LIN {X 0,Y 433.075,Z 406.489,A -85,B 0,C 180,E1 21289.378,E2 21289.378} C_VEL
LIN {X 0,Y 433.196,Z 405.398,A -85,B 0,C 180,E1 21287.416,E2 21287.416} C_VEL
LIN {X 0,Y 433.474,Z 402.273,A -85,B 0,C 180,E1 21285.29,E2 21285.29} C_VEL
LIN {X 0,Y 433.894,Z 397.242,A -85,B 0,C 180,E1 21283.265,E2 21283.265} C_VEL
LIN {X 0,Y 434.433,Z 391.164,A -85,B 0,C 180,E1 21281.517,E2 21281.517} C_VEL
LIN {X 0,Y 435.19,Z 382.602,A -85,B 0,C 180,E1 21279.675,E2 21279.675} C_VEL
LIN {X 0,Y 436.03,Z 373.053,A -85,B 0,C 180,E1 21278.086,E2 21278.086} C_VEL
LIN {X 0,Y 436.996,Z 361.523,A -85,B 0,C 180,E1 21276.573,E2 21276.573} C_VEL
LIN {X 0,Y 437.95,Z 348.916,A -85,B 0,C 180,E1 21275.283,E2 21275.283} C_VEL
LIN {X 0,Y 438.832,Z 335.315,A -85,B 0,C 180,E1 21274.2,E2 21274.2} C_VEL
LIN {X 0,Y 439.584,Z 321.029,A -85,B 0,C 180,E1 21273.335,E2 21273.335} C_VEL
LIN {X 0,Y 440.16,Z 305.307,A -85,B 0,C 180,E1 21272.665,E2 21272.665} C_VEL
LIN {X 0,Y 440.515,Z 289.237,A -85,B 0,C 180,E1 21272.235,E2 21272.235} C_VEL
LIN {X 0,Y 442.617,Z 196.385,A -85,B 0,C 180,E1 21270.394,E2 21270.394} C_VEL
LIN {X 0,Y 438.448,Z 173.54,A -85,B 0,C 180,E1 21269.604,E2 21269.604} C_VEL
LIN {X 0,Y 440.626,Z 144.172,A -85,B 0,C 180,E1 21265.541,E2 21265.541} C_VEL
LIN {X 0,Y 442.984,Z 116.613,A -85,B 0,C 180,E1 21261.65,E2 21261.65} C_VEL
LIN {X 0,Y 444.119,Z 103.787,A -85,B 0,C 180,E1 21259.806,E2 21259.806} C_VEL
LIN {X 0,Y 440.05,Z 88.666,A -85,B 0,C 180,E1 21257.044,E2 21257.044} C_VEL
LIN {X 0,Y 435.296,Z 73.845,A -85,B 0,C 180,E1 21254.092,E2 21254.092} C_VEL
LIN {X 0,Y 433.235,Z 67.94,A -85,B 0,C 180,E1 21252.767,E2 21252.767} C_VEL
LIN {X 0,Y 433.212,Z 67.828,A -85,B 0,C 180,E1 21249.03,E2 21249.03} C_VEL
LIN {X 0,Y 433.209,Z 67.837,A -85,B 0,C 180,E1 21245.297,E2 21245.297} C_VEL
LIN {X 0,Y 433.214,Z 67.833,A -85,B 0,C 180,E1 21241.587,E2 21241.587} C_VEL
LIN {X 0,Y 433.223,Z 67.833,A -85,B 0,C 180,E1 21237.924,E2 21237.924} C_VEL
LIN {X 0,Y 433.235,Z 67.831,A -85,B 0,C 180,E1 21234.172,E2 21234.172} C_VEL
LIN {X 0,Y 433.245,Z 67.831,A -85,B 0,C 180,E1 21230.435,E2 21230.435} C_VEL
LIN {X 0,Y 433.25,Z 67.833,A -85,B 0,C 180,E1 21226.657,E2 21226.657} C_VEL
LIN {X 0,Y 433.243,Z 67.831,A -85,B 0,C 180,E1 21222.818,E2 21222.818} C_VEL
LIN {X 0,Y 433.231,Z 67.83,A -85,B 0,C 180,E1 21219.04,E2 21219.04} C_VEL
LIN {X 0,Y 433.214,Z 67.833,A -85,B 0,C 180,E1 21215.308,E2 21215.308} C_VEL
LIN {X 0,Y 433.2,Z 67.836,A -85,B 0,C 180,E1 21211.611,E2 21211.611} C_VEL
LIN {X 0,Y 433.191,Z 67.837,A -85,B 0,C 180,E1 21207.896,E2 21207.896} C_VEL
LIN {X 0,Y 433.19,Z 67.836,A -85,B 0,C 180,E1 21204.108,E2 21204.108} C_VEL
LIN {X 0,Y 433.187,Z 67.839,A -85,B 0,C 180,E1 21200.256,E2 21200.256} C_VEL
LIN {X 0,Y 433.192,Z 67.835,A -85,B 0,C 180,E1 21196.542,E2 21196.542} C_VEL
LIN {X 0,Y 433.211,Z 67.832,A -85,B 0,C 180,E1 21192.912,E2 21192.912} C_VEL
LIN {X 0,Y 433.263,Z 68.081,A -85,B 0,C 180,E1 21191.105,E2 21191.105} C_VEL
LIN {X 0,Y 438.845,Z 82.472,A -85,B 0,C 180,E1 21188.603,E2 21188.603} C_VEL
LIN {X 0,Y 444.549,Z 98.48,A -85,B 0,C 180,E1 21186.153,E2 21186.153} C_VEL
LIN {X 0,Y 447.389,Z 107.578,A -85,B 0,C 180,E1 21184.895,E2 21184.895} C_VEL
LIN {X 0,Y 443.251,Z 148.715,A -85,B 0,C 180,E1 21180.876,E2 21180.876} C_VEL
LIN {X 0,Y 442.316,Z 161.133,A -85,B 0,C 180,E1 21179.733,E2 21179.733} C_VEL
LIN {X 0,Y 444.429,Z 180.599,A -85,B 0,C 180,E1 21179.248,E2 21179.248} C_VEL
LIN {X 0,Y 442.001,Z 357.769,A -85,B 0,C 180,E1 21176.343,E2 21176.343} C_VEL
LIN {X 0,Y 441.177,Z 376.273,A -85,B 0,C 180,E1 21175.815,E2 21175.815} C_VEL
LIN {X 0,Y 440.124,Z 394.053,A -85,B 0,C 180,E1 21175.068,E2 21175.068} C_VEL
LIN {X 0,Y 438.871,Z 411.762,A -85,B 0,C 180,E1 21174.068,E2 21174.068} C_VEL
LIN {X 0,Y 437.522,Z 428.981,A -85,B 0,C 180,E1 21172.82,E2 21172.82} C_VEL
LIN {X 0,Y 436.208,Z 445.015,A -85,B 0,C 180,E1 21171.375,E2 21171.375} C_VEL
LIN {X 0,Y 435.015,Z 459.816,A -85,B 0,C 180,E1 21169.748,E2 21169.748} C_VEL
LIN {X 0,Y 433.995,Z 473.598,A -85,B 0,C 180,E1 21167.92,E2 21167.92} C_VEL
LIN {X 0,Y 433.196,Z 485.958,A -85,B 0,C 180,E1 21165.943,E2 21165.943} C_VEL
LIN {X 0,Y 432.671,Z 497.125,A -85,B 0,C 180,E1 21163.771,E2 21163.771} C_VEL
LIN {X 0,Y 432.402,Z 506.213,A -85,B 0,C 180,E1 21161.606,E2 21161.606} C_VEL
LIN {X 0,Y 432.351,Z 513.891,A -85,B 0,C 180,E1 21159.317,E2 21159.317} C_VEL
LIN {X 0,Y 432.443,Z 519.752,A -85,B 0,C 180,E1 21157.04,E2 21157.04} C_VEL
LIN {X 0,Y 432.595,Z 524.105,A -85,B 0,C 180,E1 21154.641,E2 21154.641} C_VEL
LIN {X 0,Y 432.715,Z 526.668,A -85,B 0,C 180,E1 21152.252,E2 21152.252} C_VEL
LIN {X 0,Y 432.765,Z 527.51,A -85,B 0,C 180,E1 21150.001,E2 21150.001} C_VEL
LIN {X 0,Y 432.693,Z 526.696,A -85,B 0,C 180,E1 21147.617,E2 21147.617} C_VEL
LIN {X 0,Y 432.564,Z 524.137,A -85,B 0,C 180,E1 21145.228,E2 21145.228} C_VEL
LIN {X 0,Y 432.407,Z 519.767,A -85,B 0,C 180,E1 21142.828,E2 21142.828} C_VEL
LIN {X 0,Y 432.328,Z 513.478,A -85,B 0,C 180,E1 21140.416,E2 21140.416} C_VEL
LIN {X 0,Y 432.413,Z 505.642,A -85,B 0,C 180,E1 21138.125,E2 21138.125} C_VEL
LIN {X 0,Y 432.721,Z 496.365,A -85,B 0,C 180,E1 21135.96,E2 21135.96} C_VEL
LIN {X 0,Y 433.259,Z 485.712,A -85,B 0,C 180,E1 21133.924,E2 21133.924} C_VEL
LIN {X 0,Y 434.052,Z 473.719,A -85,B 0,C 180,E1 21132.022,E2 21132.022} C_VEL
LIN {X 0,Y 435.095,Z 459.77,A -85,B 0,C 180,E1 21130.188,E2 21130.188} C_VEL
LIN {X 0,Y 436.299,Z 444.783,A -85,B 0,C 180,E1 21128.562,E2 21128.562} C_VEL
LIN {X 0,Y 437.586,Z 428.819,A -85,B 0,C 180,E1 21127.144,E2 21127.144} C_VEL
LIN {X 0,Y 438.881,Z 411.866,A -85,B 0,C 180,E1 21125.935,E2 21125.935} C_VEL
LIN {X 0,Y 440.066,Z 394.468,A -85,B 0,C 180,E1 21124.967,E2 21124.967} C_VEL
LIN {X 0,Y 441.097,Z 376.307,A -85,B 0,C 180,E1 21124.217,E2 21124.217} C_VEL
LIN {X 0,Y 441.882,Z 357.278,A -85,B 0,C 180,E1 21123.69,E2 21123.69} C_VEL
LIN {X 0,Y 444.228,Z 168.638,A -85,B 0,C 180,E1 21120.613,E2 21120.613} C_VEL
LIN {X 0,Y 443.59,Z 156.452,A -85,B 0,C 180,E1 21120.348,E2 21120.348} C_VEL
LIN {X 0,Y 446.644,Z 101.681,A -85,B 0,C 180,E1 21117.321,E2 21117.321} C_VEL
LIN {X 0,Y 436.652,Z 76.57,A -85,B 0,C 180,E1 21115.06,E2 21115.06} C_VEL
LIN {X 0,Y 433.339,Z 68.369,A -85,B 0,C 180,E1 21114.246,E2 21114.246} C_VEL
LIN {X 0,Y 433.254,Z 67.833,A -85,B 0,C 180,E1 21113.952,E2 21113.952} C_VEL
LIN {X 0,Y 433.255,Z 67.829,A -85,B 0,C 180,E1 21110.094,E2 21110.094} C_VEL
LIN {X 0,Y 433.255,Z 67.829,A -85,B 0,C 180,E1 21106.247,E2 21106.247} C_VEL
LIN {X 0,Y 433.258,Z 67.83,A -85,B 0,C 180,E1 21102.366,E2 21102.366} C_VEL
LIN {X 0,Y 433.259,Z 67.826,A -85,B 0,C 180,E1 21098.528,E2 21098.528} C_VEL
LIN {X 0,Y 433.259,Z 67.822,A -85,B 0,C 180,E1 21094.751,E2 21094.751} C_VEL
LIN {X 0,Y 433.26,Z 67.824,A -85,B 0,C 180,E1 21090.857,E2 21090.857} C_VEL
LIN {X 0,Y 433.256,Z 67.822,A -85,B 0,C 180,E1 21087.03,E2 21087.03} C_VEL
LIN {X 0,Y 433.252,Z 67.819,A -85,B 0,C 180,E1 21083.243,E2 21083.243} C_VEL
LIN {X 0,Y 433.24,Z 67.823,A -85,B 0,C 180,E1 21079.55,E2 21079.55} C_VEL
LIN {X 0,Y 433.235,Z 67.827,A -85,B 0,C 180,E1 21075.771,E2 21075.771} C_VEL
LIN {X 0,Y 433.234,Z 67.83,A -85,B 0,C 180,E1 21071.988,E2 21071.988} C_VEL
LIN {X 0,Y 433.232,Z 67.829,A -85,B 0,C 180,E1 21068.093,E2 21068.093} C_VEL
LIN {X 0,Y 433.231,Z 67.825,A -85,B 0,C 180,E1 21064.235,E2 21064.235} C_VEL
LIN {X 0,Y 433.229,Z 67.822,A -85,B 0,C 180,E1 21060.396,E2 21060.396} C_VEL
LIN {X 0,Y 433.236,Z 67.829,A -85,B 0,C 180,E1 21056.692,E2 21056.692} C_VEL
LIN {X 0,Y 433.244,Z 67.833,A -85,B 0,C 180,E1 21052.902,E2 21052.902} C_VEL
LIN {X 0,Y 433.247,Z 67.829,A -85,B 0,C 180,E1 21049.091,E2 21049.091} C_VEL
LIN {X 0,Y 433.257,Z 67.824,A -85,B 0,C 180,E1 21045.294,E2 21045.294} C_VEL
LIN {X 0,Y 433.256,Z 67.824,A -85,B 0,C 180,E1 21041.429,E2 21041.429} C_VEL
LIN {X 0,Y 433.264,Z 67.81,A -85,B 0,C 180,E1 21037.618,E2 21037.618} C_VEL
LIN {X 0,Y 433.258,Z 67.826,A -85,B 0,C 180,E1 21033.698,E2 21033.698} C_VEL
LIN {X 0,Y 433.26,Z 67.809,A -85,B 0,C 180,E1 21029.926,E2 21029.926} C_VEL
LIN {X 0,Y 433.254,Z 67.83,A -85,B 0,C 180,E1 21026.048,E2 21026.048} C_VEL
LIN {X 0,Y 433.239,Z 67.832,A -85,B 0,C 180,E1 21022.295,E2 21022.295} C_VEL
LIN {X 0,Y 433.222,Z 67.83,A -85,B 0,C 180,E1 21018.595,E2 21018.595} C_VEL
LIN {X 0,Y 433.213,Z 67.834,A -85,B 0,C 180,E1 21014.882,E2 21014.882} C_VEL
LIN {X 0,Y 433.204,Z 67.837,A -85,B 0,C 180,E1 21011.13,E2 21011.13} C_VEL
LIN {X 0,Y 433.261,Z 68.1,A -85,B 0,C 180,E1 21008.676,E2 21008.676} C_VEL
LIN {X 0,Y 438.519,Z 85.922,A -85,B 0,C 180,E1 21006.292,E2 21006.292} C_VEL
LIN {X 0,Y 440.008,Z 92.89,A -85,B 0,C 180,E1 21005.41,E2 21005.41} C_VEL
LIN {X 0,Y 439.529,Z 126.207,A -85,B 0,C 180,E1 21001.699,E2 21001.699} C_VEL
LIN {X 0,Y 438.985,Z 159.572,A -85,B 0,C 180,E1 20997.981,E2 20997.981} C_VEL
LIN {X 0,Y 438.678,Z 192.545,A -85,B 0,C 180,E1 20994.455,E2 20994.455} C_VEL
LIN {X 0,Y 439.206,Z 197.779,A -85,B 0,C 180,E1 20994.332,E2 20994.332} C_VEL
LIN {X 0,Y 438.077,Z 288.666,A -85,B 0,C 180,E1 20992.826,E2 20992.826} C_VEL
LIN {X 0,Y 437.082,Z 296.35,A -85,B 0,C 180,E1 20992.742,E2 20992.742} C_VEL
LIN {X 0,Y 432.175,Z 312.347,A -85,B 0,C 180,E1 20992.59,E2 20992.59} C_VEL
LIN {X 0,Y 430.641,Z 319.881,A -85,B 0,C 180,E1 20992.382,E2 20992.382} C_VEL
LIN {X 0,Y 430.425,Z 322.967,A -85,B 0,C 180,E1 20992.254,E2 20992.254} C_VEL
LIN {X 0,Y 430.017,Z 337.032,A -85,B 0,C 180,E1 20991.481,E2 20991.481} C_VEL
LIN {X 0,Y 429.406,Z 349.966,A -85,B 0,C 180,E1 20990.512,E2 20990.512} C_VEL
LIN {X 0,Y 428.679,Z 362.566,A -85,B 0,C 180,E1 20989.27,E2 20989.27} C_VEL
LIN {X 0,Y 427.886,Z 373.856,A -85,B 0,C 180,E1 20987.824,E2 20987.824} C_VEL
LIN {X 0,Y 427.151,Z 383.064,A -85,B 0,C 180,E1 20986.312,E2 20986.312} C_VEL
LIN {X 0,Y 426.501,Z 390.945,A -85,B 0,C 180,E1 20984.665,E2 20984.665} C_VEL
LIN {X 0,Y 425.929,Z 397.841,A -85,B 0,C 180,E1 20982.747,E2 20982.747} C_VEL
LIN {X 0,Y 425.507,Z 402.946,A -85,B 0,C 180,E1 20980.697,E2 20980.697} C_VEL
LIN {X 0,Y 425.241,Z 406.026,A -85,B 0,C 180,E1 20978.654,E2 20978.654} C_VEL
LIN {X 0,Y 425.112,Z 407.274,A -85,B 0,C 180,E1 20976.617,E2 20976.617} C_VEL
LIN {X 0,Y 425.103,Z 406.761,A -85,B 0,C 180,E1 20974.586,E2 20974.586} C_VEL
LIN {X 0,Y 425.219,Z 404.234,A -85,B 0,C 180,E1 20972.425,E2 20972.425} C_VEL
LIN {X 0,Y 425.464,Z 399.9,A -85,B 0,C 180,E1 20970.403,E2 20970.403} C_VEL
LIN {X 0,Y 425.825,Z 393.939,A -85,B 0,C 180,E1 20968.519,E2 20968.519} C_VEL
LIN {X 0,Y 426.31,Z 386.487,A -85,B 0,C 180,E1 20966.772,E2 20966.772} C_VEL
LIN {X 0,Y 426.895,Z 377.575,A -85,B 0,C 180,E1 20965.162,E2 20965.162} C_VEL
LIN {X 0,Y 427.565,Z 366.546,A -85,B 0,C 180,E1 20963.622,E2 20963.622} C_VEL
LIN {X 0,Y 428.158,Z 354.829,A -85,B 0,C 180,E1 20962.35,E2 20962.35} C_VEL
LIN {X 0,Y 428.687,Z 342.994,A -85,B 0,C 180,E1 20961.347,E2 20961.347} C_VEL
LIN {X 0,Y 429.131,Z 329.341,A -85,B 0,C 180,E1 20960.477,E2 20960.477} C_VEL
LIN {X 0,Y 429.327,Z 314.736,A -85,B 0,C 180,E1 20959.825,E2 20959.825} C_VEL
LIN {X 0,Y 429.329,Z 299.926,A -85,B 0,C 180,E1 20959.423,E2 20959.423} C_VEL
LIN {X 0,Y 430.516,Z 189.532,A -85,B 0,C 180,E1 20957.56,E2 20957.56} C_VEL
LIN {X 0,Y 431.081,Z 159.552,A -85,B 0,C 180,E1 20955.629,E2 20955.629} C_VEL
LIN {X 0,Y 431.654,Z 130.351,A -85,B 0,C 180,E1 20953.653,E2 20953.653} C_VEL
LIN {X 0,Y 432.206,Z 129.541,A -85,B 0,C 180,E1 20953.433,E2 20953.433} C_VEL
LIN {X 0,Y 434.053,Z 130.583,A -85,B 0,C 180,E1 20953.161,E2 20953.161} C_VEL
LIN {X 0,Y 431.916,Z 170.793,A -85,B 0,C 180,E1 20949.928,E2 20949.928} C_VEL
LIN {X 0,Y 433.654,Z 190.939,A -85,B 0,C 180,E1 20949.44,E2 20949.44} C_VEL
LIN {X 0,Y 431.591,Z 296.803,A -85,B 0,C 180,E1 20947.438,E2 20947.438} C_VEL
LIN {X 0,Y 431.154,Z 313.161,A -85,B 0,C 180,E1 20946.871,E2 20946.871} C_VEL
LIN {X 0,Y 430.489,Z 328.565,A -85,B 0,C 180,E1 20946.064,E2 20946.064} C_VEL
LIN {X 0,Y 429.718,Z 342.273,A -85,B 0,C 180,E1 20945.092,E2 20945.092} C_VEL
LIN {X 0,Y 428.833,Z 355.782,A -85,B 0,C 180,E1 20943.853,E2 20943.853} C_VEL
LIN {X 0,Y 427.907,Z 368.637,A -85,B 0,C 180,E1 20942.324,E2 20942.324} C_VEL
LIN {X 0,Y 427.079,Z 379.255,A -85,B 0,C 180,E1 20940.705,E2 20940.705} C_VEL
LIN {X 0,Y 426.438,Z 387.604,A -85,B 0,C 180,E1 20939.103,E2 20939.103} C_VEL
LIN {X 0,Y 425.856,Z 395.37,A -85,B 0,C 180,E1 20937.155,E2 20937.155} C_VEL
LIN {X 0,Y 425.493,Z 400.746,A -85,B 0,C 180,E1 20935.333,E2 20935.333} C_VEL
LIN {X 0,Y 425.248,Z 404.826,A -85,B 0,C 180,E1 20933.3,E2 20933.3} C_VEL
LIN {X 0,Y 425.139,Z 407.07,A -85,B 0,C 180,E1 20931.274,E2 20931.274} C_VEL
LIN {X 0,Y 425.165,Z 407.601,A -85,B 0,C 180,E1 20929.173,E2 20929.173} C_VEL
LIN {X 0,Y 425.304,Z 406.351,A -85,B 0,C 180,E1 20927.18,E2 20927.18} C_VEL
LIN {X 0,Y 425.607,Z 403.261,A -85,B 0,C 180,E1 20925.096,E2 20925.096} C_VEL
LIN {X 0,Y 426.062,Z 398.275,A -85,B 0,C 180,E1 20923.071,E2 20923.071} C_VEL
LIN {X 0,Y 426.687,Z 391.722,A -85,B 0,C 180,E1 20921.184,E2 20921.184} C_VEL
LIN {X 0,Y 427.515,Z 383.155,A -85,B 0,C 180,E1 20919.332,E2 20919.332} C_VEL
LIN {X 0,Y 428.437,Z 373.304,A -85,B 0,C 180,E1 20917.694,E2 20917.694} C_VEL
LIN {X 0,Y 429.449,Z 361.862,A -85,B 0,C 180,E1 20916.191,E2 20916.191} C_VEL
LIN {X 0,Y 430.51,Z 348.756,A -85,B 0,C 180,E1 20914.844,E2 20914.844} C_VEL
LIN {X 0,Y 431.43,Z 335.21,A -85,B 0,C 180,E1 20913.769,E2 20913.769} C_VEL
LIN {X 0,Y 432.234,Z 320.637,A -85,B 0,C 180,E1 20912.891,E2 20912.891} C_VEL
LIN {X 0,Y 432.865,Z 304.237,A -85,B 0,C 180,E1 20912.199,E2 20912.199} C_VEL
LIN {X 0,Y 433.284,Z 285.362,A -85,B 0,C 180,E1 20911.729,E2 20911.729} C_VEL
LIN {X 0,Y 435.428,Z 197.571,A -85,B 0,C 180,E1 20909.949,E2 20909.949} C_VEL
LIN {X 0,Y 430.996,Z 173.326,A -85,B 0,C 180,E1 20909.081,E2 20909.081} C_VEL
LIN {X 0,Y 433.342,Z 144.216,A -85,B 0,C 180,E1 20904.976,E2 20904.976} C_VEL
LIN {X 0,Y 435.85,Z 117.318,A -85,B 0,C 180,E1 20901.111,E2 20901.111} C_VEL
LIN {X 0,Y 436.789,Z 106.47,A -85,B 0,C 180,E1 20899.525,E2 20899.525} C_VEL
LIN {X 0,Y 432.67,Z 91.123,A -85,B 0,C 180,E1 20896.652,E2 20896.652} C_VEL
LIN {X 0,Y 428.146,Z 77.113,A -85,B 0,C 180,E1 20893.781,E2 20893.781} C_VEL
LIN {X 0,Y 425.328,Z 68.949,A -85,B 0,C 180,E1 20891.939,E2 20891.939} C_VEL
LIN {X 0,Y 425.321,Z 68.817,A -85,B 0,C 180,E1 20888.109,E2 20888.109} C_VEL
LIN {X 0,Y 425.312,Z 68.82,A -85,B 0,C 180,E1 20884.315,E2 20884.315} C_VEL
LIN {X 0,Y 425.322,Z 68.819,A -85,B 0,C 180,E1 20880.404,E2 20880.404} C_VEL
LIN {X 0,Y 425.308,Z 68.821,A -85,B 0,C 180,E1 20876.496,E2 20876.496} C_VEL
LIN {X 0,Y 425.32,Z 68.819,A -85,B 0,C 180,E1 20872.571,E2 20872.571} C_VEL
LIN {X 0,Y 425.307,Z 68.821,A -85,B 0,C 180,E1 20868.611,E2 20868.611} C_VEL
LIN {X 0,Y 425.311,Z 68.821,A -85,B 0,C 180,E1 20864.734,E2 20864.734} C_VEL
LIN {X 0,Y 425.305,Z 68.819,A -85,B 0,C 180,E1 20860.784,E2 20860.784} C_VEL
LIN {X 0,Y 425.307,Z 68.818,A -85,B 0,C 180,E1 20856.884,E2 20856.884} C_VEL
LIN {X 0,Y 425.3,Z 68.819,A -85,B 0,C 180,E1 20853.001,E2 20853.001} C_VEL
LIN {X 0,Y 425.294,Z 68.82,A -85,B 0,C 180,E1 20849.169,E2 20849.169} C_VEL
LIN {X 0,Y 425.282,Z 68.822,A -85,B 0,C 180,E1 20845.323,E2 20845.323} C_VEL
LIN {X 0,Y 425.272,Z 68.825,A -85,B 0,C 180,E1 20841.529,E2 20841.529} C_VEL
LIN {X 0,Y 425.25,Z 68.827,A -85,B 0,C 180,E1 20837.925,E2 20837.925} C_VEL
LIN {X 0,Y 425.253,Z 68.824,A -85,B 0,C 180,E1 20834.104,E2 20834.104} C_VEL
LIN {X 0,Y 425.296,Z 69.092,A -85,B 0,C 180,E1 20831.982,E2 20831.982} C_VEL
LIN {X 0,Y 430.877,Z 83.146,A -85,B 0,C 180,E1 20829.4,E2 20829.4} C_VEL
LIN {X 0,Y 436.843,Z 99.589,A -85,B 0,C 180,E1 20826.766,E2 20826.766} C_VEL
LIN {X 0,Y 440.209,Z 110.166,A -85,B 0,C 180,E1 20825.235,E2 20825.235} C_VEL
LIN {X 0,Y 435.706,Z 152.651,A -85,B 0,C 180,E1 20821.01,E2 20821.01} C_VEL
LIN {X 0,Y 435.023,Z 161.252,A -85,B 0,C 180,E1 20820.209,E2 20820.209} C_VEL
LIN {X 0,Y 437.229,Z 181.414,A -85,B 0,C 180,E1 20819.693,E2 20819.693} C_VEL
LIN {X 0,Y 434.628,Z 357.34,A -85,B 0,C 180,E1 20816.756,E2 20816.756} C_VEL
LIN {X 0,Y 433.759,Z 375.802,A -85,B 0,C 180,E1 20816.219,E2 20816.219} C_VEL
LIN {X 0,Y 432.644,Z 393.542,A -85,B 0,C 180,E1 20815.459,E2 20815.459} C_VEL
LIN {X 0,Y 431.315,Z 411.168,A -85,B 0,C 180,E1 20814.444,E2 20814.444} C_VEL
LIN {X 0,Y 429.924,Z 427.831,A -85,B 0,C 180,E1 20813.217,E2 20813.217} C_VEL
LIN {X 0,Y 428.548,Z 443.615,A -85,B 0,C 180,E1 20811.776,E2 20811.776} C_VEL
LIN {X 0,Y 427.263,Z 458.477,A -85,B 0,C 180,E1 20810.122,E2 20810.122} C_VEL
LIN {X 0,Y 426.191,Z 471.87,A -85,B 0,C 180,E1 20808.323,E2 20808.323} C_VEL
LIN {X 0,Y 425.295,Z 484.717,A -85,B 0,C 180,E1 20806.247,E2 20806.247} C_VEL
LIN {X 0,Y 424.714,Z 495.919,A -85,B 0,C 180,E1 20804.034,E2 20804.034} C_VEL
LIN {X 0,Y 424.425,Z 505.036,A -85,B 0,C 180,E1 20801.828,E2 20801.828} C_VEL
LIN {X 0,Y 424.371,Z 512.736,A -85,B 0,C 180,E1 20799.494,E2 20799.494} C_VEL
LIN {X 0,Y 424.474,Z 518.615,A -85,B 0,C 180,E1 20797.173,E2 20797.173} C_VEL
LIN {X 0,Y 424.648,Z 522.983,A -85,B 0,C 180,E1 20794.728,E2 20794.728} C_VEL
LIN {X 0,Y 424.776,Z 525.476,A -85,B 0,C 180,E1 20792.429,E2 20792.429} C_VEL
LIN {X 0,Y 424.842,Z 526.401,A -85,B 0,C 180,E1 20790.001,E2 20790.001} C_VEL
LIN {X 0,Y 424.763,Z 525.58,A -85,B 0,C 180,E1 20787.573,E2 20787.573} C_VEL
LIN {X 0,Y 424.613,Z 523.005,A -85,B 0,C 180,E1 20785.138,E2 20785.138} C_VEL
LIN {X 0,Y 424.442,Z 518.61,A -85,B 0,C 180,E1 20782.693,E2 20782.693} C_VEL
LIN {X 0,Y 424.35,Z 512.711,A -85,B 0,C 180,E1 20780.371,E2 20780.371} C_VEL
LIN {X 0,Y 424.428,Z 504.945,A -85,B 0,C 180,E1 20778.037,E2 20778.037} C_VEL
LIN {X 0,Y 424.744,Z 495.736,A -85,B 0,C 180,E1 20775.83,E2 20775.83} C_VEL
LIN {X 0,Y 425.311,Z 485.158,A -85,B 0,C 180,E1 20773.756,E2 20773.756} C_VEL
LIN {X 0,Y 426.145,Z 473.25,A -85,B 0,C 180,E1 20771.818,E2 20771.818} C_VEL
LIN {X 0,Y 427.242,Z 459.383,A -85,B 0,C 180,E1 20769.951,E2 20769.951} C_VEL
LIN {X 0,Y 428.506,Z 444.483,A -85,B 0,C 180,E1 20768.296,E2 20768.296} C_VEL
LIN {X 0,Y 429.926,Z 427.783,A -85,B 0,C 180,E1 20766.786,E2 20766.786} C_VEL
LIN {X 0,Y 431.214,Z 411.814,A -85,B 0,C 180,E1 20765.625,E2 20765.625} C_VEL
LIN {X 0,Y 432.456,Z 394.611,A -85,B 0,C 180,E1 20764.641,E2 20764.641} C_VEL
LIN {X 0,Y 433.541,Z 376.567,A -85,B 0,C 180,E1 20763.874,E2 20763.874} C_VEL
LIN {X 0,Y 434.371,Z 357.859,A -85,B 0,C 180,E1 20763.336,E2 20763.336} C_VEL
LIN {X 0,Y 436.872,Z 168.968,A -85,B 0,C 180,E1 20760.199,E2 20760.199} C_VEL
LIN {X 0,Y 436.235,Z 156.887,A -85,B 0,C 180,E1 20759.938,E2 20759.938} C_VEL
LIN {X 0,Y 439.399,Z 104.304,A -85,B 0,C 180,E1 20756.985,E2 20756.985} C_VEL
LIN {X 0,Y 429.21,Z 78.595,A -85,B 0,C 180,E1 20754.621,E2 20754.621} C_VEL
LIN {X 0,Y 425.41,Z 69.401,A -85,B 0,C 180,E1 20753.683,E2 20753.683} C_VEL
LIN {X 0,Y 425.318,Z 68.855,A -85,B 0,C 180,E1 20753.506,E2 20753.506} C_VEL
LIN {X 0,Y 425.316,Z 68.818,A -85,B 0,C 180,E1 20749.612,E2 20749.612} C_VEL
LIN {X 0,Y 425.315,Z 68.817,A -85,B 0,C 180,E1 20745.719,E2 20745.719} C_VEL
LIN {X 0,Y 425.317,Z 68.817,A -85,B 0,C 180,E1 20741.825,E2 20741.825} C_VEL
LIN {X 0,Y 425.318,Z 68.816,A -85,B 0,C 180,E1 20738.019,E2 20738.019} C_VEL
LIN {X 0,Y 425.317,Z 68.818,A -85,B 0,C 180,E1 20734.16,E2 20734.16} C_VEL
LIN {X 0,Y 425.325,Z 68.817,A -85,B 0,C 180,E1 20730.359,E2 20730.359} C_VEL
LIN {X 0,Y 425.319,Z 68.815,A -85,B 0,C 180,E1 20726.529,E2 20726.529} C_VEL
LIN {X 0,Y 425.324,Z 68.81,A -85,B 0,C 180,E1 20722.677,E2 20722.677} C_VEL
LIN {X 0,Y 425.322,Z 68.809,A -85,B 0,C 180,E1 20718.788,E2 20718.788} C_VEL
LIN {X 0,Y 425.323,Z 68.813,A -85,B 0,C 180,E1 20714.95,E2 20714.95} C_VEL
LIN {X 0,Y 425.32,Z 68.818,A -85,B 0,C 180,E1 20711.114,E2 20711.114} C_VEL
LIN {X 0,Y 425.325,Z 68.815,A -85,B 0,C 180,E1 20707.249,E2 20707.249} C_VEL
LIN {X 0,Y 425.315,Z 68.812,A -85,B 0,C 180,E1 20703.369,E2 20703.369} C_VEL
LIN {X 0,Y 425.321,Z 68.806,A -85,B 0,C 180,E1 20699.461,E2 20699.461} C_VEL
LIN {X 0,Y 425.314,Z 68.814,A -85,B 0,C 180,E1 20695.55,E2 20695.55} C_VEL
LIN {X 0,Y 425.309,Z 68.817,A -85,B 0,C 180,E1 20691.755,E2 20691.755} C_VEL
LIN {X 0,Y 425.3,Z 68.818,A -85,B 0,C 180,E1 20687.922,E2 20687.922} C_VEL
LIN {X 0,Y 425.29,Z 68.818,A -85,B 0,C 180,E1 20684.174,E2 20684.174} C_VEL
LIN {X 0,Y 425.287,Z 68.819,A -85,B 0,C 180,E1 20680.354,E2 20680.354} C_VEL
LIN {X 0,Y 425.279,Z 68.793,A -85,B 0,C 180,E1 20676.588,E2 20676.588} C_VEL
LIN {X 0,Y 425.279,Z 68.821,A -85,B 0,C 180,E1 20672.706,E2 20672.706} C_VEL
LIN {X 0,Y 425.276,Z 68.81,A -85,B 0,C 180,E1 20668.844,E2 20668.844} C_VEL
LIN {X 0,Y 425.276,Z 68.81,A -85,B 0,C 180,E1 20664.993,E2 20664.993} C_VEL
LIN {X 0,Y 425.272,Z 68.822,A -85,B 0,C 180,E1 20661.095,E2 20661.095} C_VEL
LIN {X 0,Y 425.277,Z 68.822,A -85,B 0,C 180,E1 20657.38,E2 20657.38} C_VEL
LIN {X 0,Y 425.283,Z 68.817,A -85,B 0,C 180,E1 20653.604,E2 20653.604} C_VEL
LIN {X 0,Y 425.298,Z 68.817,A -85,B 0,C 180,E1 20649.925,E2 20649.925} C_VEL
LIN {X 0,Y 425.304,Z 69.093,A -85,B 0,C 180,E1 20649.182,E2 20649.182} C_VEL
LIN {X 0,Y 430.618,Z 86.53,A -85,B 0,C 180,E1 20646.8,E2 20646.8} C_VEL
LIN {X 0,Y 432.615,Z 95.017,A -85,B 0,C 180,E1 20645.701,E2 20645.701} C_VEL
LIN {X 0,Y 432.08,Z 128.838,A -85,B 0,C 180,E1 20641.912,E2 20641.912} C_VEL
LIN {X 0,Y 431.492,Z 162.665,A -85,B 0,C 180,E1 20638.133,E2 20638.133} C_VEL
LIN {X 0,Y 431.22,Z 193.709,A -85,B 0,C 180,E1 20634.817,E2 20634.817} C_VEL
LIN {X 0,Y 431.74,Z 198.821,A -85,B 0,C 180,E1 20634.699,E2 20634.699} C_VEL
LIN {X 0,Y 430.576,Z 304.253,A -85,B 0,C 180,E1 20632.893,E2 20632.893} C_VEL
LIN {X 0,Y 430.495,Z 319.294,A -85,B 0,C 180,E1 20632.414,E2 20632.414} C_VEL
LIN {X 0,Y 430.425,Z 322.967,A -85,B 0,C 180,E1 20632.254,E2 20632.254} C_VEL
LIN {X 0,Y 429.319,Z 330.3,A -85,B 0,C 180,E1 20631.943,E2 20631.943} C_VEL
LIN {X 0,Y 424.622,Z 343.262,A -85,B 0,C 180,E1 20631.323,E2 20631.323} C_VEL
LIN {X 0,Y 422.152,Z 350.932,A -85,B 0,C 180,E1 20630.81,E2 20630.81} C_VEL
LIN {X 0,Y 421.602,Z 354.646,A -85,B 0,C 180,E1 20630.492,E2 20630.492} C_VEL
LIN {X 0,Y 420.794,Z 367.109,A -85,B 0,C 180,E1 20629.14,E2 20629.14} C_VEL
LIN {X 0,Y 420,Z 377.165,A -85,B 0,C 180,E1 20627.74,E2 20627.74} C_VEL
LIN {X 0,Y 419.251,Z 385.949,A -85,B 0,C 180,E1 20626.201,E2 20626.201} C_VEL
LIN {X 0,Y 418.533,Z 393.939,A -85,B 0,C 180,E1 20624.385,E2 20624.385} C_VEL
LIN {X 0,Y 417.955,Z 400.278,A -85,B 0,C 180,E1 20622.432,E2 20622.432} C_VEL
LIN {X 0,Y 417.562,Z 404.661,A -85,B 0,C 180,E1 20620.484,E2 20620.484} C_VEL
LIN {X 0,Y 417.305,Z 407.461,A -85,B 0,C 180,E1 20618.403,E2 20618.403} C_VEL
LIN {X 0,Y 417.179,Z 408.427,A -85,B 0,C 180,E1 20616.19,E2 20616.19} C_VEL
LIN {X 0,Y 417.194,Z 407.361,A -85,B 0,C 180,E1 20613.984,E2 20613.984} C_VEL
LIN {X 0,Y 417.341,Z 404.489,A -85,B 0,C 180,E1 20611.921,E2 20611.921} C_VEL
LIN {X 0,Y 417.609,Z 400.087,A -85,B 0,C 180,E1 20609.999,E2 20609.999} C_VEL
LIN {X 0,Y 418.026,Z 393.808,A -85,B 0,C 180,E1 20608.08,E2 20608.08} C_VEL
LIN {X 0,Y 418.565,Z 385.948,A -85,B 0,C 180,E1 20606.301,E2 20606.301} C_VEL
LIN {X 0,Y 419.203,Z 376.524,A -85,B 0,C 180,E1 20604.662,E2 20604.662} C_VEL
LIN {X 0,Y 419.856,Z 366.186,A -85,B 0,C 180,E1 20603.248,E2 20603.248} C_VEL
LIN {X 0,Y 420.501,Z 353.897,A -85,B 0,C 180,E1 20601.935,E2 20601.935} C_VEL
LIN {X 0,Y 421.098,Z 340.426,A -85,B 0,C 180,E1 20600.845,E2 20600.845} C_VEL
LIN {X 0,Y 421.495,Z 326.627,A -85,B 0,C 180,E1 20600.027,E2 20600.027} C_VEL
LIN {X 0,Y 421.648,Z 312.384,A -85,B 0,C 180,E1 20599.443,E2 20599.443} C_VEL
LIN {X 0,Y 421.603,Z 295.98,A -85,B 0,C 180,E1 20599.06,E2 20599.06} C_VEL
LIN {X 0,Y 422.859,Z 190.683,A -85,B 0,C 180,E1 20597.261,E2 20597.261} C_VEL
LIN {X 0,Y 423.297,Z 176.085,A -85,B 0,C 180,E1 20596.336,E2 20596.336} C_VEL
LIN {X 0,Y 423.969,Z 136.619,A -85,B 0,C 180,E1 20593.701,E2 20593.701} C_VEL
LIN {X 0,Y 424.417,Z 135.354,A -85,B 0,C 180,E1 20593.472,E2 20593.472} C_VEL
LIN {X 0,Y 425.897,Z 135.981,A -85,B 0,C 180,E1 20593.215,E2 20593.215} C_VEL
LIN {X 0,Y 426.359,Z 136.325,A -85,B 0,C 180,E1 20593.155,E2 20593.155} C_VEL
LIN {X 0,Y 424.462,Z 170.682,A -85,B 0,C 180,E1 20590.359,E2 20590.359} C_VEL
LIN {X 0,Y 426.25,Z 191.647,A -85,B 0,C 180,E1 20589.837,E2 20589.837} C_VEL
LIN {X 0,Y 424.067,Z 297.435,A -85,B 0,C 180,E1 20587.794,E2 20587.794} C_VEL
LIN {X 0,Y 423.612,Z 313.551,A -85,B 0,C 180,E1 20587.226,E2 20587.226} C_VEL
LIN {X 0,Y 422.948,Z 328.267,A -85,B 0,C 180,E1 20586.451,E2 20586.451} C_VEL
LIN {X 0,Y 422.125,Z 342.477,A -85,B 0,C 180,E1 20585.445,E2 20585.445} C_VEL
LIN {X 0,Y 421.171,Z 356.29,A -85,B 0,C 180,E1 20584.167,E2 20584.167} C_VEL
LIN {X 0,Y 420.219,Z 368.837,A -85,B 0,C 180,E1 20582.663,E2 20582.663} C_VEL
LIN {X 0,Y 419.406,Z 378.784,A -85,B 0,C 180,E1 20581.163,E2 20581.163} C_VEL
LIN {X 0,Y 418.612,Z 388.496,A -85,B 0,C 180,E1 20579.302,E2 20579.302} C_VEL
LIN {X 0,Y 417.997,Z 396.186,A -85,B 0,C 180,E1 20577.352,E2 20577.352} C_VEL
LIN {X 0,Y 417.594,Z 401.811,A -85,B 0,C 180,E1 20575.426,E2 20575.426} C_VEL
LIN {X 0,Y 417.334,Z 405.877,A -85,B 0,C 180,E1 20573.375,E2 20573.375} C_VEL
LIN {X 0,Y 417.22,Z 408.12,A -85,B 0,C 180,E1 20571.376,E2 20571.376} C_VEL
LIN {X 0,Y 417.247,Z 408.724,A -85,B 0,C 180,E1 20569.141,E2 20569.141} C_VEL
LIN {X 0,Y 417.397,Z 407.513,A -85,B 0,C 180,E1 20567.132,E2 20567.132} C_VEL
LIN {X 0,Y 417.71,Z 404.591,A -85,B 0,C 180,E1 20565.078,E2 20565.078} C_VEL
LIN {X 0,Y 418.158,Z 400.09,A -85,B 0,C 180,E1 20563.146,E2 20563.146} C_VEL
LIN {X 0,Y 418.846,Z 393.439,A -85,B 0,C 180,E1 20561.124,E2 20561.124} C_VEL
LIN {X 0,Y 419.697,Z 385.143,A -85,B 0,C 180,E1 20559.262,E2 20559.262} C_VEL
LIN {X 0,Y 420.635,Z 376.009,A -85,B 0,C 180,E1 20557.655,E2 20557.655} C_VEL
LIN {X 0,Y 421.778,Z 364.082,A -85,B 0,C 180,E1 20556.009,E2 20556.009} C_VEL
LIN {X 0,Y 422.889,Z 351.247,A -85,B 0,C 180,E1 20554.634,E2 20554.634} C_VEL
LIN {X 0,Y 423.903,Z 337.672,A -85,B 0,C 180,E1 20553.5,E2 20553.5} C_VEL
LIN {X 0,Y 424.822,Z 322.329,A -85,B 0,C 180,E1 20552.534,E2 20552.534} C_VEL
LIN {X 0,Y 425.498,Z 305.996,A -85,B 0,C 180,E1 20551.819,E2 20551.819} C_VEL
LIN {X 0,Y 425.908,Z 289.31,A -85,B 0,C 180,E1 20551.367,E2 20551.367} C_VEL
LIN {X 0,Y 428.272,Z 198.78,A -85,B 0,C 180,E1 20549.489,E2 20549.489} C_VEL
LIN {X 0,Y 423.6,Z 173.348,A -85,B 0,C 180,E1 20548.554,E2 20548.554} C_VEL
LIN {X 0,Y 426.079,Z 144.478,A -85,B 0,C 180,E1 20544.425,E2 20544.425} C_VEL
LIN {X 0,Y 428.804,Z 117.432,A -85,B 0,C 180,E1 20540.473,E2 20540.473} C_VEL
LIN {X 0,Y 429.572,Z 109.541,A -85,B 0,C 180,E1 20539.3,E2 20539.3} C_VEL
LIN {X 0,Y 425.708,Z 94.924,A -85,B 0,C 180,E1 20536.511,E2 20536.511} C_VEL
LIN {X 0,Y 421.256,Z 80.961,A -85,B 0,C 180,E1 20533.591,E2 20533.591} C_VEL
LIN {X 0,Y 417.356,Z 69.94,A -85,B 0,C 180,E1 20531.015,E2 20531.015} C_VEL
LIN {X 0,Y 417.337,Z 69.813,A -85,B 0,C 180,E1 20527.157,E2 20527.157} C_VEL
LIN {X 0,Y 417.333,Z 69.814,A -85,B 0,C 180,E1 20523.297,E2 20523.297} C_VEL
LIN {X 0,Y 417.33,Z 69.811,A -85,B 0,C 180,E1 20519.451,E2 20519.451} C_VEL
LIN {X 0,Y 417.33,Z 69.812,A -85,B 0,C 180,E1 20515.603,E2 20515.603} C_VEL
LIN {X 0,Y 417.329,Z 69.812,A -85,B 0,C 180,E1 20511.735,E2 20511.735} C_VEL
LIN {X 0,Y 417.332,Z 69.81,A -85,B 0,C 180,E1 20507.969,E2 20507.969} C_VEL
LIN {X 0,Y 417.346,Z 69.809,A -85,B 0,C 180,E1 20504.293,E2 20504.293} C_VEL
LIN {X 0,Y 417.361,Z 69.811,A -85,B 0,C 180,E1 20500.549,E2 20500.549} C_VEL
LIN {X 0,Y 417.365,Z 69.809,A -85,B 0,C 180,E1 20496.717,E2 20496.717} C_VEL
LIN {X 0,Y 417.358,Z 69.809,A -85,B 0,C 180,E1 20492.769,E2 20492.769} C_VEL
LIN {X 0,Y 417.367,Z 69.807,A -85,B 0,C 180,E1 20488.999,E2 20488.999} C_VEL
LIN {X 0,Y 417.357,Z 69.811,A -85,B 0,C 180,E1 20485.018,E2 20485.018} C_VEL
LIN {X 0,Y 417.367,Z 69.81,A -85,B 0,C 180,E1 20481.123,E2 20481.123} C_VEL
LIN {X 0,Y 417.351,Z 69.812,A -85,B 0,C 180,E1 20477.313,E2 20477.313} C_VEL
LIN {X 0,Y 417.35,Z 69.805,A -85,B 0,C 180,E1 20473.439,E2 20473.439} C_VEL
LIN {X 0,Y 417.402,Z 70.272,A -85,B 0,C 180,E1 20472.868,E2 20472.868} C_VEL
LIN {X 0,Y 423.109,Z 84.192,A -85,B 0,C 180,E1 20470.176,E2 20470.176} C_VEL
LIN {X 0,Y 429.15,Z 100.807,A -85,B 0,C 180,E1 20467.394,E2 20467.394} C_VEL
LIN {X 0,Y 433.063,Z 112.987,A -85,B 0,C 180,E1 20465.579,E2 20465.579} C_VEL
LIN {X 0,Y 428.514,Z 152.97,A -85,B 0,C 180,E1 20461.512,E2 20461.512} C_VEL
LIN {X 0,Y 427.809,Z 161.554,A -85,B 0,C 180,E1 20460.703,E2 20460.703} C_VEL
LIN {X 0,Y 430.056,Z 182.277,A -85,B 0,C 180,E1 20460.153,E2 20460.153} C_VEL
LIN {X 0,Y 427.307,Z 356.603,A -85,B 0,C 180,E1 20457.195,E2 20457.195} C_VEL
LIN {X 0,Y 426.393,Z 375.051,A -85,B 0,C 180,E1 20456.651,E2 20456.651} C_VEL
LIN {X 0,Y 425.189,Z 393.093,A -85,B 0,C 180,E1 20455.863,E2 20455.863} C_VEL
LIN {X 0,Y 423.779,Z 410.611,A -85,B 0,C 180,E1 20454.833,E2 20454.833} C_VEL
LIN {X 0,Y 422.311,Z 427.212,A -85,B 0,C 180,E1 20453.587,E2 20453.587} C_VEL
LIN {X 0,Y 420.916,Z 442.238,A -85,B 0,C 180,E1 20452.192,E2 20452.192} C_VEL
LIN {X 0,Y 419.525,Z 457.186,A -85,B 0,C 180,E1 20450.505,E2 20450.505} C_VEL
LIN {X 0,Y 418.329,Z 471.083,A -85,B 0,C 180,E1 20448.608,E2 20448.608} C_VEL
LIN {X 0,Y 417.401,Z 483.483,A -85,B 0,C 180,E1 20446.563,E2 20446.563} C_VEL
LIN {X 0,Y 416.765,Z 494.725,A -85,B 0,C 180,E1 20444.307,E2 20444.307} C_VEL
LIN {X 0,Y 416.45,Z 503.865,A -85,B 0,C 180,E1 20442.058,E2 20442.058} C_VEL
LIN {X 0,Y 416.388,Z 511.584,A -85,B 0,C 180,E1 20439.678,E2 20439.678} C_VEL
LIN {X 0,Y 416.505,Z 517.482,A -85,B 0,C 180,E1 20437.311,E2 20437.311} C_VEL
LIN {X 0,Y 416.68,Z 521.685,A -85,B 0,C 180,E1 20434.957,E2 20434.957} C_VEL
LIN {X 0,Y 416.845,Z 524.364,A -85,B 0,C 180,E1 20432.476,E2 20432.476} C_VEL
LIN {X 0,Y 416.919,Z 525.29,A -85,B 0,C 180,E1 20430.001,E2 20430.001} C_VEL
LIN {X 0,Y 416.834,Z 524.461,A -85,B 0,C 180,E1 20427.526,E2 20427.526} C_VEL
LIN {X 0,Y 416.661,Z 521.867,A -85,B 0,C 180,E1 20425.045,E2 20425.045} C_VEL
LIN {X 0,Y 416.475,Z 517.393,A -85,B 0,C 180,E1 20422.53,E2 20422.53} C_VEL
LIN {X 0,Y 416.37,Z 511.508,A -85,B 0,C 180,E1 20420.184,E2 20420.184} C_VEL
LIN {X 0,Y 416.457,Z 503.7,A -85,B 0,C 180,E1 20417.804,E2 20417.804} C_VEL
LIN {X 0,Y 416.802,Z 494.436,A -85,B 0,C 180,E1 20415.554,E2 20415.554} C_VEL
LIN {X 0,Y 417.453,Z 483.255,A -85,B 0,C 180,E1 20413.346,E2 20413.346} C_VEL
LIN {X 0,Y 418.386,Z 470.826,A -85,B 0,C 180,E1 20411.324,E2 20411.324} C_VEL
LIN {X 0,Y 419.594,Z 456.672,A -85,B 0,C 180,E1 20409.424,E2 20409.424} C_VEL
LIN {X 0,Y 420.915,Z 442.093,A -85,B 0,C 180,E1 20407.811,E2 20407.811} C_VEL
LIN {X 0,Y 422.355,Z 425.967,A -85,B 0,C 180,E1 20406.352,E2 20406.352} C_VEL
LIN {X 0,Y 423.727,Z 409.633,A -85,B 0,C 180,E1 20405.166,E2 20405.166} C_VEL
LIN {X 0,Y 425.057,Z 392.013,A -85,B 0,C 180,E1 20404.168,E2 20404.168} C_VEL
LIN {X 0,Y 426.194,Z 373.462,A -85,B 0,C 180,E1 20403.399,E2 20403.399} C_VEL
LIN {X 0,Y 426.976,Z 354.676,A -85,B 0,C 180,E1 20402.889,E2 20402.889} C_VEL
LIN {X 0,Y 429.544,Z 169.625,A -85,B 0,C 180,E1 20399.783,E2 20399.783} C_VEL
LIN {X 0,Y 428.925,Z 156.081,A -85,B 0,C 180,E1 20399.459,E2 20399.459} C_VEL
LIN {X 0,Y 432.004,Z 106.521,A -85,B 0,C 180,E1 20396.601,E2 20396.601} C_VEL
LIN {X 0,Y 422.303,Z 82.074,A -85,B 0,C 180,E1 20394.301,E2 20394.301} C_VEL
LIN {X 0,Y 417.451,Z 70.311,A -85,B 0,C 180,E1 20393.075,E2 20393.075} C_VEL
LIN {X 0,Y 417.377,Z 69.83,A -85,B 0,C 180,E1 20392.868,E2 20392.868} C_VEL
LIN {X 0,Y 417.372,Z 69.81,A -85,B 0,C 180,E1 20388.977,E2 20388.977} C_VEL
LIN {X 0,Y 417.373,Z 69.808,A -85,B 0,C 180,E1 20385.035,E2 20385.035} C_VEL
LIN {X 0,Y 417.368,Z 69.803,A -85,B 0,C 180,E1 20381.208,E2 20381.208} C_VEL
LIN {X 0,Y 417.368,Z 69.808,A -85,B 0,C 180,E1 20377.307,E2 20377.307} C_VEL
LIN {X 0,Y 417.365,Z 69.808,A -85,B 0,C 180,E1 20373.435,E2 20373.435} C_VEL
LIN {X 0,Y 417.364,Z 69.807,A -85,B 0,C 180,E1 20369.571,E2 20369.571} C_VEL
LIN {X 0,Y 417.362,Z 69.808,A -85,B 0,C 180,E1 20365.697,E2 20365.697} C_VEL
LIN {X 0,Y 417.361,Z 69.808,A -85,B 0,C 180,E1 20361.797,E2 20361.797} C_VEL
LIN {X 0,Y 417.358,Z 69.807,A -85,B 0,C 180,E1 20357.857,E2 20357.857} C_VEL
LIN {X 0,Y 417.356,Z 69.802,A -85,B 0,C 180,E1 20354.002,E2 20354.002} C_VEL
LIN {X 0,Y 417.356,Z 69.799,A -85,B 0,C 180,E1 20350.069,E2 20350.069} C_VEL
LIN {X 0,Y 417.354,Z 69.805,A -85,B 0,C 180,E1 20346.183,E2 20346.183} C_VEL
LIN {X 0,Y 417.354,Z 69.808,A -85,B 0,C 180,E1 20342.334,E2 20342.334} C_VEL
LIN {X 0,Y 417.354,Z 69.809,A -85,B 0,C 180,E1 20338.49,E2 20338.49} C_VEL
LIN {X 0,Y 417.354,Z 69.803,A -85,B 0,C 180,E1 20334.639,E2 20334.639} C_VEL
LIN {X 0,Y 417.361,Z 69.801,A -85,B 0,C 180,E1 20330.902,E2 20330.902} C_VEL
LIN {X 0,Y 417.37,Z 69.804,A -85,B 0,C 180,E1 20327.127,E2 20327.127} C_VEL
LIN {X 0,Y 417.373,Z 69.807,A -85,B 0,C 180,E1 20323.293,E2 20323.293} C_VEL
LIN {X 0,Y 417.374,Z 69.807,A -85,B 0,C 180,E1 20319.381,E2 20319.381} C_VEL
LIN {X 0,Y 417.372,Z 69.781,A -85,B 0,C 180,E1 20315.516,E2 20315.516} C_VEL
LIN {X 0,Y 417.381,Z 69.801,A -85,B 0,C 180,E1 20311.684,E2 20311.684} C_VEL
LIN {X 0,Y 417.379,Z 69.802,A -85,B 0,C 180,E1 20307.871,E2 20307.871} C_VEL
LIN {X 0,Y 417.371,Z 69.792,A -85,B 0,C 180,E1 20304.06,E2 20304.06} C_VEL
LIN {X 0,Y 417.367,Z 69.799,A -85,B 0,C 180,E1 20300.235,E2 20300.235} C_VEL
LIN {X 0,Y 417.362,Z 69.8,A -85,B 0,C 180,E1 20296.373,E2 20296.373} C_VEL
LIN {X 0,Y 417.345,Z 69.803,A -85,B 0,C 180,E1 20292.65,E2 20292.65} C_VEL
LIN {X 0,Y 417.38,Z 70.064,A -85,B 0,C 180,E1 20289.716,E2 20289.716} C_VEL
LIN {X 0,Y 423.007,Z 88.169,A -85,B 0,C 180,E1 20287.196,E2 20287.196} C_VEL
LIN {X 0,Y 425.252,Z 97.229,A -85,B 0,C 180,E1 20285.999,E2 20285.999} C_VEL
LIN {X 0,Y 424.658,Z 131.412,A -85,B 0,C 180,E1 20282.147,E2 20282.147} C_VEL
LIN {X 0,Y 424.031,Z 165.157,A -85,B 0,C 180,E1 20278.366,E2 20278.366} C_VEL
LIN {X 0,Y 423.753,Z 194.667,A -85,B 0,C 180,E1 20275.202,E2 20275.202} C_VEL
LIN {X 0,Y 424.292,Z 199.862,A -85,B 0,C 180,E1 20275.078,E2 20275.078} C_VEL
LIN {X 0,Y 423.057,Z 304.88,A -85,B 0,C 180,E1 20273.25,E2 20273.25} C_VEL
LIN {X 0,Y 422.971,Z 320.161,A -85,B 0,C 180,E1 20272.76,E2 20272.76} C_VEL
LIN {X 0,Y 422.592,Z 334.651,A -85,B 0,C 180,E1 20272.024,E2 20272.024} C_VEL
LIN {X 0,Y 422,Z 347.594,A -85,B 0,C 180,E1 20271.107,E2 20271.107} C_VEL
LIN {X 0,Y 421.602,Z 354.646,A -85,B 0,C 180,E1 20270.492,E2 20270.492} C_VEL
LIN {X 0,Y 420.27,Z 361.005,A -85,B 0,C 180,E1 20269.909,E2 20269.909} C_VEL
LIN {X 0,Y 415.263,Z 372.031,A -85,B 0,C 180,E1 20268.803,E2 20268.803} C_VEL
LIN {X 0,Y 412.652,Z 378.228,A -85,B 0,C 180,E1 20267.995,E2 20267.995} C_VEL
LIN {X 0,Y 412.046,Z 381.099,A -85,B 0,C 180,E1 20267.534,E2 20267.534} C_VEL
LIN {X 0,Y 411.215,Z 390.033,A -85,B 0,C 180,E1 20265.801,E2 20265.801} C_VEL
LIN {X 0,Y 410.463,Z 397.768,A -85,B 0,C 180,E1 20263.81,E2 20263.81} C_VEL
LIN {X 0,Y 409.889,Z 403.635,A -85,B 0,C 180,E1 20261.68,E2 20261.68} C_VEL
LIN {X 0,Y 409.512,Z 407.377,A -85,B 0,C 180,E1 20259.556,E2 20259.556} C_VEL
LIN {X 0,Y 409.316,Z 409.176,A -85,B 0,C 180,E1 20257.579,E2 20257.579} C_VEL
LIN {X 0,Y 409.243,Z 409.387,A -85,B 0,C 180,E1 20255.467,E2 20255.467} C_VEL
LIN {X 0,Y 409.306,Z 407.631,A -85,B 0,C 180,E1 20253.22,E2 20253.22} C_VEL
LIN {X 0,Y 409.516,Z 404.08,A -85,B 0,C 180,E1 20251.118,E2 20251.118} C_VEL
LIN {X 0,Y 409.853,Z 398.968,A -85,B 0,C 180,E1 20249.16,E2 20249.16} C_VEL
LIN {X 0,Y 410.322,Z 392.456,A -85,B 0,C 180,E1 20247.345,E2 20247.345} C_VEL
LIN {X 0,Y 410.946,Z 383.824,A -85,B 0,C 180,E1 20245.534,E2 20245.534} C_VEL
LIN {X 0,Y 411.6,Z 374.434,A -85,B 0,C 180,E1 20244.003,E2 20244.003} C_VEL
LIN {X 0,Y 412.288,Z 363.685,A -85,B 0,C 180,E1 20242.614,E2 20242.614} C_VEL
LIN {X 0,Y 412.933,Z 351.246,A -85,B 0,C 180,E1 20241.365,E2 20241.365} C_VEL
LIN {X 0,Y 413.484,Z 338.536,A -85,B 0,C 180,E1 20240.394,E2 20240.394} C_VEL
LIN {X 0,Y 413.845,Z 325.072,A -85,B 0,C 180,E1 20239.63,E2 20239.63} C_VEL
LIN {X 0,Y 413.967,Z 309.464,A -85,B 0,C 180,E1 20239.043,E2 20239.043} C_VEL
LIN {X 0,Y 414.036,Z 277.659,A -85,B 0,C 180,E1 20238.439,E2 20238.439} C_VEL
LIN {X 0,Y 415.214,Z 191.837,A -85,B 0,C 180,E1 20236.952,E2 20236.952} C_VEL
LIN {X 0,Y 415.653,Z 180.187,A -85,B 0,C 180,E1 20236.222,E2 20236.222} C_VEL
LIN {X 0,Y 416.359,Z 141.961,A -85,B 0,C 180,E1 20233.645,E2 20233.645} C_VEL
LIN {X 0,Y 416.929,Z 141.115,A -85,B 0,C 180,E1 20233.418,E2 20233.418} C_VEL
LIN {X 0,Y 418.663,Z 142.071,A -85,B 0,C 180,E1 20233.149,E2 20233.149} C_VEL
LIN {X 0,Y 417.027,Z 170.578,A -85,B 0,C 180,E1 20230.805,E2 20230.805} C_VEL
LIN {X 0,Y 418.864,Z 192.429,A -85,B 0,C 180,E1 20230.247,E2 20230.247} C_VEL
LIN {X 0,Y 416.56,Z 298.031,A -85,B 0,C 180,E1 20228.163,E2 20228.163} C_VEL
LIN {X 0,Y 416.074,Z 314.307,A -85,B 0,C 180,E1 20227.577,E2 20227.577} C_VEL
LIN {X 0,Y 415.34,Z 329.697,A -85,B 0,C 180,E1 20226.746,E2 20226.746} C_VEL
LIN {X 0,Y 414.47,Z 343.752,A -85,B 0,C 180,E1 20225.72,E2 20225.72} C_VEL
LIN {X 0,Y 413.474,Z 357.449,A -85,B 0,C 180,E1 20224.421,E2 20224.421} C_VEL
LIN {X 0,Y 412.441,Z 370.355,A -85,B 0,C 180,E1 20222.836,E2 20222.836} C_VEL
LIN {X 0,Y 411.502,Z 381.122,A -85,B 0,C 180,E1 20221.141,E2 20221.141} C_VEL
LIN {X 0,Y 410.755,Z 389.784,A -85,B 0,C 180,E1 20219.419,E2 20219.419} C_VEL
LIN {X 0,Y 410.103,Z 397.552,A -85,B 0,C 180,E1 20217.397,E2 20217.397} C_VEL
LIN {X 0,Y 409.659,Z 403.301,A -85,B 0,C 180,E1 20215.338,E2 20215.338} C_VEL
LIN {X 0,Y 409.402,Z 407.278,A -85,B 0,C 180,E1 20213.232,E2 20213.232} C_VEL
LIN {X 0,Y 409.291,Z 409.481,A -85,B 0,C 180,E1 20210.973,E2 20210.973} C_VEL
LIN {X 0,Y 409.336,Z 409.801,A -85,B 0,C 180,E1 20208.923,E2 20208.923} C_VEL
LIN {X 0,Y 409.545,Z 408.268,A -85,B 0,C 180,E1 20206.681,E2 20206.681} C_VEL
LIN {X 0,Y 409.907,Z 404.999,A -85,B 0,C 180,E1 20204.581,E2 20204.581} C_VEL
LIN {X 0,Y 410.495,Z 399.717,A -85,B 0,C 180,E1 20202.436,E2 20202.436} C_VEL
LIN {X 0,Y 411.262,Z 392.756,A -85,B 0,C 180,E1 20200.45,E2 20200.45} C_VEL
LIN {X 0,Y 412.197,Z 384.427,A -85,B 0,C 180,E1 20198.641,E2 20198.641} C_VEL
LIN {X 0,Y 413.337,Z 373.879,A -85,B 0,C 180,E1 20196.864,E2 20196.864} C_VEL
LIN {X 0,Y 414.502,Z 362.095,A -85,B 0,C 180,E1 20195.317,E2 20195.317} C_VEL
LIN {X 0,Y 415.656,Z 349.349,A -85,B 0,C 180,E1 20193.998,E2 20193.998} C_VEL
LIN {X 0,Y 416.759,Z 334.77,A -85,B 0,C 180,E1 20192.834,E2 20192.834} C_VEL
LIN {X 0,Y 417.639,Z 319.718,A -85,B 0,C 180,E1 20191.944,E2 20191.944} C_VEL
LIN {X 0,Y 418.277,Z 304.345,A -85,B 0,C 180,E1 20191.302,E2 20191.302} C_VEL
LIN {X 0,Y 418.829,Z 283.232,A -85,B 0,C 180,E1 20190.775,E2 20190.775} C_VEL
LIN {X 0,Y 421.161,Z 199.979,A -85,B 0,C 180,E1 20189.006,E2 20189.006} C_VEL
LIN {X 0,Y 416.244,Z 173.141,A -85,B 0,C 180,E1 20187.983,E2 20187.983} C_VEL
LIN {X 0,Y 418.922,Z 144.378,A -85,B 0,C 180,E1 20183.789,E2 20183.789} C_VEL
LIN {X 0,Y 421.842,Z 117.441,A -85,B 0,C 180,E1 20179.784,E2 20179.784} C_VEL
LIN {X 0,Y 422.391,Z 112.668,A -85,B 0,C 180,E1 20179.067,E2 20179.067} C_VEL
LIN {X 0,Y 418.475,Z 97.794,A -85,B 0,C 180,E1 20176.159,E2 20176.159} C_VEL
LIN {X 0,Y 414.034,Z 83.656,A -85,B 0,C 180,E1 20173.121,E2 20173.121} C_VEL
LIN {X 0,Y 410.188,Z 73.372,A -85,B 0,C 180,E1 20170.676,E2 20170.676} C_VEL
LIN {X 0,Y 409.442,Z 70.877,A -85,B 0,C 180,E1 20169.985,E2 20169.985} C_VEL
LIN {X 0,Y 409.439,Z 70.799,A -85,B 0,C 180,E1 20166.169,E2 20166.169} C_VEL
LIN {X 0,Y 409.433,Z 70.798,A -85,B 0,C 180,E1 20162.24,E2 20162.24} C_VEL
LIN {X 0,Y 409.433,Z 70.798,A -85,B 0,C 180,E1 20158.321,E2 20158.321} C_VEL
LIN {X 0,Y 409.432,Z 70.797,A -85,B 0,C 180,E1 20154.395,E2 20154.395} C_VEL
LIN {X 0,Y 409.429,Z 70.798,A -85,B 0,C 180,E1 20150.583,E2 20150.583} C_VEL
LIN {X 0,Y 409.431,Z 70.798,A -85,B 0,C 180,E1 20146.586,E2 20146.586} C_VEL
LIN {X 0,Y 409.426,Z 70.799,A -85,B 0,C 180,E1 20142.667,E2 20142.667} C_VEL
LIN {X 0,Y 409.43,Z 70.796,A -85,B 0,C 180,E1 20138.812,E2 20138.812} C_VEL
LIN {X 0,Y 409.422,Z 70.797,A -85,B 0,C 180,E1 20134.854,E2 20134.854} C_VEL
LIN {X 0,Y 409.428,Z 70.796,A -85,B 0,C 180,E1 20130.924,E2 20130.924} C_VEL
LIN {X 0,Y 409.42,Z 70.798,A -85,B 0,C 180,E1 20127.003,E2 20127.003} C_VEL
LIN {X 0,Y 409.417,Z 70.802,A -85,B 0,C 180,E1 20123.075,E2 20123.075} C_VEL
LIN {X 0,Y 409.426,Z 70.798,A -85,B 0,C 180,E1 20119.205,E2 20119.205} C_VEL
LIN {X 0,Y 409.413,Z 70.793,A -85,B 0,C 180,E1 20115.29,E2 20115.29} C_VEL
LIN {X 0,Y 409.429,Z 71.125,A -85,B 0,C 180,E1 20113.911,E2 20113.911} C_VEL
LIN {X 0,Y 414.409,Z 83.369,A -85,B 0,C 180,E1 20111.379,E2 20111.379} C_VEL
LIN {X 0,Y 419.273,Z 95.942,A -85,B 0,C 180,E1 20109.083,E2 20109.083} C_VEL
LIN {X 0,Y 424.542,Z 111.468,A -85,B 0,C 180,E1 20106.572,E2 20106.572} C_VEL
LIN {X 0,Y 425.852,Z 116.329,A -85,B 0,C 180,E1 20105.868,E2 20105.868} C_VEL
LIN {X 0,Y 420.836,Z 158.405,A -85,B 0,C 180,E1 20101.514,E2 20101.514} C_VEL
LIN {X 0,Y 420.632,Z 161.829,A -85,B 0,C 180,E1 20101.218,E2 20101.218} C_VEL
LIN {X 0,Y 422.945,Z 183.213,A -85,B 0,C 180,E1 20100.635,E2 20100.635} C_VEL
LIN {X 0,Y 420.293,Z 344.01,A -85,B 0,C 180,E1 20097.884,E2 20097.884} C_VEL
LIN {X 0,Y 419.702,Z 363.354,A -85,B 0,C 180,E1 20097.46,E2 20097.46} C_VEL
LIN {X 0,Y 418.578,Z 381.848,A -85,B 0,C 180,E1 20096.8,E2 20096.8} C_VEL
LIN {X 0,Y 417.237,Z 399.075,A -85,B 0,C 180,E1 20095.935,E2 20095.935} C_VEL
LIN {X 0,Y 415.7,Z 416.339,A -85,B 0,C 180,E1 20094.794,E2 20094.794} C_VEL
LIN {X 0,Y 414.095,Z 432.95,A -85,B 0,C 180,E1 20093.404,E2 20093.404} C_VEL
LIN {X 0,Y 412.516,Z 448.73,A -85,B 0,C 180,E1 20091.768,E2 20091.768} C_VEL
LIN {X 0,Y 411.142,Z 462.913,A -85,B 0,C 180,E1 20089.98,E2 20089.98} C_VEL
LIN {X 0,Y 409.957,Z 476.561,A -85,B 0,C 180,E1 20087.898,E2 20087.898} C_VEL
LIN {X 0,Y 409.085,Z 488.687,A -85,B 0,C 180,E1 20085.637,E2 20085.637} C_VEL
LIN {X 0,Y 408.595,Z 498.91,A -85,B 0,C 180,E1 20083.299,E2 20083.299} C_VEL
LIN {X 0,Y 408.401,Z 507.46,A -85,B 0,C 180,E1 20080.867,E2 20080.867} C_VEL
LIN {X 0,Y 408.467,Z 514.109,A -85,B 0,C 180,E1 20078.447,E2 20078.447} C_VEL
LIN {X 0,Y 408.641,Z 519.007,A -85,B 0,C 180,E1 20076.04,E2 20076.04} C_VEL
LIN {X 0,Y 408.843,Z 522.261,A -85,B 0,C 180,E1 20073.647,E2 20073.647} C_VEL
LIN {X 0,Y 408.972,Z 523.934,A -85,B 0,C 180,E1 20071.262,E2 20071.262} C_VEL
LIN {X 0,Y 408.972,Z 524.027,A -85,B 0,C 180,E1 20068.88,E2 20068.88} C_VEL
LIN {X 0,Y 408.825,Z 522.404,A -85,B 0,C 180,E1 20066.355,E2 20066.355} C_VEL
LIN {X 0,Y 408.607,Z 518.99,A -85,B 0,C 180,E1 20063.82,E2 20063.82} C_VEL
LIN {X 0,Y 408.434,Z 513.693,A -85,B 0,C 180,E1 20061.271,E2 20061.271} C_VEL
LIN {X 0,Y 408.4,Z 506.854,A -85,B 0,C 180,E1 20058.849,E2 20058.849} C_VEL
LIN {X 0,Y 408.644,Z 498.031,A -85,B 0,C 180,E1 20056.416,E2 20056.416} C_VEL
LIN {X 0,Y 409.173,Z 487.657,A -85,B 0,C 180,E1 20054.118,E2 20054.118} C_VEL
LIN {X 0,Y 410.039,Z 475.759,A -85,B 0,C 180,E1 20051.961,E2 20051.961} C_VEL
LIN {X 0,Y 411.198,Z 462.289,A -85,B 0,C 180,E1 20049.951,E2 20049.951} C_VEL
LIN {X 0,Y 412.573,Z 447.668,A -85,B 0,C 180,E1 20048.154,E2 20048.154} C_VEL
LIN {X 0,Y 414.082,Z 431.931,A -85,B 0,C 180,E1 20046.572,E2 20046.572} C_VEL
LIN {X 0,Y 415.568,Z 415.671,A -85,B 0,C 180,E1 20045.253,E2 20045.253} C_VEL
LIN {X 0,Y 417.022,Z 398.002,A -85,B 0,C 180,E1 20044.129,E2 20044.129} C_VEL
LIN {X 0,Y 418.289,Z 379.984,A -85,B 0,C 180,E1 20043.273,E2 20043.273} C_VEL
LIN {X 0,Y 419.262,Z 361.67,A -85,B 0,C 180,E1 20042.668,E2 20042.668} C_VEL
LIN {X 0,Y 419.772,Z 339.126,A -85,B 0,C 180,E1 20042.221,E2 20042.221} C_VEL
LIN {X 0,Y 422.242,Z 170.343,A -85,B 0,C 180,E1 20039.353,E2 20039.353} C_VEL
LIN {X 0,Y 421.604,Z 156.646,A -85,B 0,C 180,E1 20039.029,E2 20039.029} C_VEL
LIN {X 0,Y 424.798,Z 109.23,A -85,B 0,C 180,E1 20036.258,E2 20036.258} C_VEL
LIN {X 0,Y 414.889,Z 84.123,A -85,B 0,C 180,E1 20033.836,E2 20033.836} C_VEL
LIN {X 0,Y 409.526,Z 71.334,A -85,B 0,C 180,E1 20032.463,E2 20032.463} C_VEL
LIN {X 0,Y 409.44,Z 70.807,A -85,B 0,C 180,E1 20032.199,E2 20032.199} C_VEL
LIN {X 0,Y 409.441,Z 70.795,A -85,B 0,C 180,E1 20028.353,E2 20028.353} C_VEL
LIN {X 0,Y 409.44,Z 70.798,A -85,B 0,C 180,E1 20024.496,E2 20024.496} C_VEL
LIN {X 0,Y 409.444,Z 70.792,A -85,B 0,C 180,E1 20020.509,E2 20020.509} C_VEL
LIN {X 0,Y 409.441,Z 70.798,A -85,B 0,C 180,E1 20016.545,E2 20016.545} C_VEL
LIN {X 0,Y 409.442,Z 70.795,A -85,B 0,C 180,E1 20012.6,E2 20012.6} C_VEL
LIN {X 0,Y 409.448,Z 70.792,A -85,B 0,C 180,E1 20008.595,E2 20008.595} C_VEL
LIN {X 0,Y 409.443,Z 70.795,A -85,B 0,C 180,E1 20004.682,E2 20004.682} C_VEL
LIN {X 0,Y 409.444,Z 70.797,A -85,B 0,C 180,E1 20000.732,E2 20000.732} C_VEL
LIN {X 0,Y 409.444,Z 70.796,A -85,B 0,C 180,E1 19996.747,E2 19996.747} C_VEL
LIN {X 0,Y 409.442,Z 70.792,A -85,B 0,C 180,E1 19992.839,E2 19992.839} C_VEL
LIN {X 0,Y 409.441,Z 70.786,A -85,B 0,C 180,E1 19988.85,E2 19988.85} C_VEL
LIN {X 0,Y 409.438,Z 70.787,A -85,B 0,C 180,E1 19984.903,E2 19984.903} C_VEL
LIN {X 0,Y 409.445,Z 70.791,A -85,B 0,C 180,E1 19980.979,E2 19980.979} C_VEL
LIN {X 0,Y 409.436,Z 70.799,A -85,B 0,C 180,E1 19977.06,E2 19977.06} C_VEL
LIN {X 0,Y 409.444,Z 70.796,A -85,B 0,C 180,E1 19973.127,E2 19973.127} C_VEL
LIN {X 0,Y 409.435,Z 70.793,A -85,B 0,C 180,E1 19969.161,E2 19969.161} C_VEL
LIN {X 0,Y 409.437,Z 70.79,A -85,B 0,C 180,E1 19965.242,E2 19965.242} C_VEL
LIN {X 0,Y 409.435,Z 70.791,A -85,B 0,C 180,E1 19961.342,E2 19961.342} C_VEL
LIN {X 0,Y 409.435,Z 70.772,A -85,B 0,C 180,E1 19957.455,E2 19957.455} C_VEL
LIN {X 0,Y 409.44,Z 70.793,A -85,B 0,C 180,E1 19953.612,E2 19953.612} C_VEL
LIN {X 0,Y 409.448,Z 70.772,A -85,B 0,C 180,E1 19949.798,E2 19949.798} C_VEL
LIN {X 0,Y 409.435,Z 70.791,A -85,B 0,C 180,E1 19945.828,E2 19945.828} C_VEL
LIN {X 0,Y 409.439,Z 70.802,A -85,B 0,C 180,E1 19941.841,E2 19941.841} C_VEL
LIN {X 0,Y 409.435,Z 70.799,A -85,B 0,C 180,E1 19937.932,E2 19937.932} C_VEL
LIN {X 0,Y 409.434,Z 70.797,A -85,B 0,C 180,E1 19934.103,E2 19934.103} C_VEL
LIN {X 0,Y 409.473,Z 71.04,A -85,B 0,C 180,E1 19930.273,E2 19930.273} C_VEL
LIN {X 0,Y 415.551,Z 90.329,A -85,B 0,C 180,E1 19927.539,E2 19927.539} C_VEL
LIN {X 0,Y 417.908,Z 100.271,A -85,B 0,C 180,E1 19926.223,E2 19926.223} C_VEL
LIN {X 0,Y 417.257,Z 134.14,A -85,B 0,C 180,E1 19922.38,E2 19922.38} C_VEL
LIN {X 0,Y 416.575,Z 168.419,A -85,B 0,C 180,E1 19918.529,E2 19918.529} C_VEL
LIN {X 0,Y 416.314,Z 195.701,A -85,B 0,C 180,E1 19915.599,E2 19915.599} C_VEL
LIN {X 0,Y 416.864,Z 200.775,A -85,B 0,C 180,E1 19915.474,E2 19915.474} C_VEL
LIN {X 0,Y 415.556,Z 305.429,A -85,B 0,C 180,E1 19913.623,E2 19913.623} C_VEL
LIN {X 0,Y 415.465,Z 321.016,A -85,B 0,C 180,E1 19913.121,E2 19913.121} C_VEL
LIN {X 0,Y 415.061,Z 335.585,A -85,B 0,C 180,E1 19912.37,E2 19912.37} C_VEL
LIN {X 0,Y 414.435,Z 348.578,A -85,B 0,C 180,E1 19911.437,E2 19911.437} C_VEL
LIN {X 0,Y 413.695,Z 360.493,A -85,B 0,C 180,E1 19910.32,E2 19910.32} C_VEL
LIN {X 0,Y 412.804,Z 372.469,A -85,B 0,C 180,E1 19908.864,E2 19908.864} C_VEL
LIN {X 0,Y 412.046,Z 381.099,A -85,B 0,C 180,E1 19907.534,E2 19907.534} C_VEL
LIN {X 0,Y 410.636,Z 385.965,A -85,B 0,C 180,E1 19906.704,E2 19906.704} C_VEL
LIN {X 0,Y 405.576,Z 394.087,A -85,B 0,C 180,E1 19905.168,E2 19905.168} C_VEL
LIN {X 0,Y 403.032,Z 398.375,A -85,B 0,C 180,E1 19904.123,E2 19904.123} C_VEL
LIN {X 0,Y 402.497,Z 400.23,A -85,B 0,C 180,E1 19903.557,E2 19903.557} C_VEL
LIN {X 0,Y 401.975,Z 405.173,A -85,B 0,C 180,E1 19901.622,E2 19901.622} C_VEL
LIN {X 0,Y 401.588,Z 408.751,A -85,B 0,C 180,E1 19899.457,E2 19899.457} C_VEL
LIN {X 0,Y 401.37,Z 410.487,A -85,B 0,C 180,E1 19897.154,E2 19897.154} C_VEL
LIN {X 0,Y 401.313,Z 410.253,A -85,B 0,C 180,E1 19895.001,E2 19895.001} C_VEL
LIN {X 0,Y 401.404,Z 408.259,A -85,B 0,C 180,E1 19892.854,E2 19892.854} C_VEL
LIN {X 0,Y 401.654,Z 404.423,A -85,B 0,C 180,E1 19890.712,E2 19890.712} C_VEL
LIN {X 0,Y 402.074,Z 398.528,A -85,B 0,C 180,E1 19888.574,E2 19888.574} C_VEL
LIN {X 0,Y 402.655,Z 390.852,A -85,B 0,C 180,E1 19886.582,E2 19886.582} C_VEL
LIN {X 0,Y 403.31,Z 382.19,A -85,B 0,C 180,E1 19884.879,E2 19884.879} C_VEL
LIN {X 0,Y 404.038,Z 372.086,A -85,B 0,C 180,E1 19883.32,E2 19883.32} C_VEL
LIN {X 0,Y 404.767,Z 360.38,A -85,B 0,C 180,E1 19881.905,E2 19881.905} C_VEL
LIN {X 0,Y 405.438,Z 347.408,A -85,B 0,C 180,E1 19880.703,E2 19880.703} C_VEL
LIN {X 0,Y 405.957,Z 334.128,A -85,B 0,C 180,E1 19879.785,E2 19879.785} C_VEL
LIN {X 0,Y 406.232,Z 319.904,A -85,B 0,C 180,E1 19879.079,E2 19879.079} C_VEL
LIN {X 0,Y 406.27,Z 304.61,A -85,B 0,C 180,E1 19878.608,E2 19878.608} C_VEL
LIN {X 0,Y 407.58,Z 193.006,A -85,B 0,C 180,E1 19876.631,E2 19876.631} C_VEL
LIN {X 0,Y 408.048,Z 182.968,A -85,B 0,C 180,E1 19876.012,E2 19876.012} C_VEL
LIN {X 0,Y 408.67,Z 148.109,A -85,B 0,C 180,E1 19873.658,E2 19873.658} C_VEL
LIN {X 0,Y 409.188,Z 147.023,A -85,B 0,C 180,E1 19873.424,E2 19873.424} C_VEL
LIN {X 0,Y 410.923,Z 147.974,A -85,B 0,C 180,E1 19873.132,E2 19873.132} C_VEL
LIN {X 0,Y 409.602,Z 170.487,A -85,B 0,C 180,E1 19871.262,E2 19871.262} C_VEL
LIN {X 0,Y 411.493,Z 193.186,A -85,B 0,C 180,E1 19870.668,E2 19870.668} C_VEL
LIN {X 0,Y 409.068,Z 298.47,A -85,B 0,C 180,E1 19868.547,E2 19868.547} C_VEL
LIN {X 0,Y 408.56,Z 314.682,A -85,B 0,C 180,E1 19867.956,E2 19867.956} C_VEL
LIN {X 0,Y 407.776,Z 330.393,A -85,B 0,C 180,E1 19867.095,E2 19867.095} C_VEL
LIN {X 0,Y 406.887,Z 344.139,A -85,B 0,C 180,E1 19866.079,E2 19866.079} C_VEL
LIN {X 0,Y 405.845,Z 357.807,A -85,B 0,C 180,E1 19864.772,E2 19864.772} C_VEL
LIN {X 0,Y 404.794,Z 370.289,A -85,B 0,C 180,E1 19863.232,E2 19863.232} C_VEL
LIN {X 0,Y 403.85,Z 380.685,A -85,B 0,C 180,E1 19861.617,E2 19861.617} C_VEL
LIN {X 0,Y 402.97,Z 390.333,A -85,B 0,C 180,E1 19859.709,E2 19859.709} C_VEL
LIN {X 0,Y 402.271,Z 398.109,A -85,B 0,C 180,E1 19857.682,E2 19857.682} C_VEL
LIN {X 0,Y 401.813,Z 403.759,A -85,B 0,C 180,E1 19855.705,E2 19855.705} C_VEL
LIN {X 0,Y 401.501,Z 408.071,A -85,B 0,C 180,E1 19853.474,E2 19853.474} C_VEL
LIN {X 0,Y 401.37,Z 410.394,A -85,B 0,C 180,E1 19851.297,E2 19851.297} C_VEL
LIN {X 0,Y 401.416,Z 410.965,A -85,B 0,C 180,E1 19849.002,E2 19849.002} C_VEL
LIN {X 0,Y 401.617,Z 409.613,A -85,B 0,C 180,E1 19846.792,E2 19846.792} C_VEL
LIN {X 0,Y 401.998,Z 406.581,A -85,B 0,C 180,E1 19844.655,E2 19844.655} C_VEL
LIN {X 0,Y 402.598,Z 401.489,A -85,B 0,C 180,E1 19842.472,E2 19842.472} C_VEL
LIN {X 0,Y 403.38,Z 394.996,A -85,B 0,C 180,E1 19840.498,E2 19840.498} C_VEL
LIN {X 0,Y 404.409,Z 386.437,A -85,B 0,C 180,E1 19838.539,E2 19838.539} C_VEL
LIN {X 0,Y 405.539,Z 376.617,A -85,B 0,C 180,E1 19836.807,E2 19836.807} C_VEL
LIN {X 0,Y 406.766,Z 365.31,A -85,B 0,C 180,E1 19835.224,E2 19835.224} C_VEL
LIN {X 0,Y 408.043,Z 352.282,A -85,B 0,C 180,E1 19833.796,E2 19833.796} C_VEL
LIN {X 0,Y 409.122,Z 339.407,A -85,B 0,C 180,E1 19832.691,E2 19832.691} C_VEL
LIN {X 0,Y 410.147,Z 324.317,A -85,B 0,C 180,E1 19831.702,E2 19831.702} C_VEL
LIN {X 0,Y 410.907,Z 308.379,A -85,B 0,C 180,E1 19830.964,E2 19830.964} C_VEL
LIN {X 0,Y 411.384,Z 292.152,A -85,B 0,C 180,E1 19830.485,E2 19830.485} C_VEL
LIN {X 0,Y 414.102,Z 201.299,A -85,B 0,C 180,E1 19828.511,E2 19828.511} C_VEL
LIN {X 0,Y 408.937,Z 173.091,A -85,B 0,C 180,E1 19827.405,E2 19827.405} C_VEL
LIN {X 0,Y 411.731,Z 145.003,A -85,B 0,C 180,E1 19823.243,E2 19823.243} C_VEL
LIN {X 0,Y 414.881,Z 117.863,A -85,B 0,C 180,E1 19819.133,E2 19819.133} C_VEL
LIN {X 0,Y 415.04,Z 115.065,A -85,B 0,C 180,E1 19818.688,E2 19818.688} C_VEL
LIN {X 0,Y 411.263,Z 100.704,A -85,B 0,C 180,E1 19815.801,E2 19815.801} C_VEL
LIN {X 0,Y 407.188,Z 87.584,A -85,B 0,C 180,E1 19812.912,E2 19812.912} C_VEL
LIN {X 0,Y 402.679,Z 75.127,A -85,B 0,C 180,E1 19809.865,E2 19809.865} C_VEL
LIN {X 0,Y 401.476,Z 71.913,A -85,B 0,C 180,E1 19808.955,E2 19808.955} C_VEL
LIN {X 0,Y 401.456,Z 71.794,A -85,B 0,C 180,E1 19805.144,E2 19805.144} C_VEL
LIN {X 0,Y 401.455,Z 71.789,A -85,B 0,C 180,E1 19801.285,E2 19801.285} C_VEL
LIN {X 0,Y 401.453,Z 71.79,A -85,B 0,C 180,E1 19797.288,E2 19797.288} C_VEL
LIN {X 0,Y 401.45,Z 71.791,A -85,B 0,C 180,E1 19793.422,E2 19793.422} C_VEL
LIN {X 0,Y 401.449,Z 71.791,A -85,B 0,C 180,E1 19789.525,E2 19789.525} C_VEL
LIN {X 0,Y 401.445,Z 71.788,A -85,B 0,C 180,E1 19785.578,E2 19785.578} C_VEL
LIN {X 0,Y 401.446,Z 71.786,A -85,B 0,C 180,E1 19781.611,E2 19781.611} C_VEL
LIN {X 0,Y 401.44,Z 71.791,A -85,B 0,C 180,E1 19777.754,E2 19777.754} C_VEL
LIN {X 0,Y 401.443,Z 71.792,A -85,B 0,C 180,E1 19773.842,E2 19773.842} C_VEL
LIN {X 0,Y 401.438,Z 71.793,A -85,B 0,C 180,E1 19769.959,E2 19769.959} C_VEL
LIN {X 0,Y 401.437,Z 71.793,A -85,B 0,C 180,E1 19766.038,E2 19766.038} C_VEL
LIN {X 0,Y 401.434,Z 71.792,A -85,B 0,C 180,E1 19762.033,E2 19762.033} C_VEL
LIN {X 0,Y 401.431,Z 71.795,A -85,B 0,C 180,E1 19758.124,E2 19758.124} C_VEL
LIN {X 0,Y 401.492,Z 71.976,A -85,B 0,C 180,E1 19755.048,E2 19755.048} C_VEL
LIN {X 0,Y 402.924,Z 75.569,A -85,B 0,C 180,E1 19754.18,E2 19754.18} C_VEL
LIN {X 0,Y 408.785,Z 89.72,A -85,B 0,C 180,E1 19751.226,E2 19751.226} C_VEL
LIN {X 0,Y 414.266,Z 104.721,A -85,B 0,C 180,E1 19748.514,E2 19748.514} C_VEL
LIN {X 0,Y 418.775,Z 118.814,A -85,B 0,C 180,E1 19746.266,E2 19746.266} C_VEL
LIN {X 0,Y 413.451,Z 160.95,A -85,B 0,C 180,E1 19741.817,E2 19741.817} C_VEL
LIN {X 0,Y 415.874,Z 183.703,A -85,B 0,C 180,E1 19741.142,E2 19741.142} C_VEL
LIN {X 0,Y 412.744,Z 355.363,A -85,B 0,C 180,E1 19738.119,E2 19738.119} C_VEL
LIN {X 0,Y 411.75,Z 373.732,A -85,B 0,C 180,E1 19737.558,E2 19737.558} C_VEL
LIN {X 0,Y 410.406,Z 391.672,A -85,B 0,C 180,E1 19736.751,E2 19736.751} C_VEL
LIN {X 0,Y 408.785,Z 409.663,A -85,B 0,C 180,E1 19735.654,E2 19735.654} C_VEL
LIN {X 0,Y 407.152,Z 426.09,A -85,B 0,C 180,E1 19734.367,E2 19734.367} C_VEL
LIN {X 0,Y 405.51,Z 441.659,A -85,B 0,C 180,E1 19732.852,E2 19732.852} C_VEL
LIN {X 0,Y 403.913,Z 456.764,A -85,B 0,C 180,E1 19731.055,E2 19731.055} C_VEL
LIN {X 0,Y 402.6,Z 470.028,A -85,B 0,C 180,E1 19729.137,E2 19729.137} C_VEL
LIN {X 0,Y 401.526,Z 482.585,A -85,B 0,C 180,E1 19726.939,E2 19726.939} C_VEL
LIN {X 0,Y 400.818,Z 493.582,A -85,B 0,C 180,E1 19724.594,E2 19724.594} C_VEL
LIN {X 0,Y 400.467,Z 503.016,A -85,B 0,C 180,E1 19722.107,E2 19722.107} C_VEL
LIN {X 0,Y 400.436,Z 510.827,A -85,B 0,C 180,E1 19719.486,E2 19719.486} C_VEL
LIN {X 0,Y 400.605,Z 516.34,A -85,B 0,C 180,E1 19717.026,E2 19717.026} C_VEL
LIN {X 0,Y 400.847,Z 520.344,A -85,B 0,C 180,E1 19714.436,E2 19714.436} C_VEL
LIN {X 0,Y 401.02,Z 522.464,A -85,B 0,C 180,E1 19712.001,E2 19712.001} C_VEL
LIN {X 0,Y 401.066,Z 523.01,A -85,B 0,C 180,E1 19709.573,E2 19709.573} C_VEL
LIN {X 0,Y 400.957,Z 521.981,A -85,B 0,C 180,E1 19707.142,E2 19707.142} C_VEL
LIN {X 0,Y 400.749,Z 519.359,A -85,B 0,C 180,E1 19704.704,E2 19704.704} C_VEL
LIN {X 0,Y 400.534,Z 515.089,A -85,B 0,C 180,E1 19702.254,E2 19702.254} C_VEL
LIN {X 0,Y 400.409,Z 509.076,A -85,B 0,C 180,E1 19699.789,E2 19699.789} C_VEL
LIN {X 0,Y 400.526,Z 501.167,A -85,B 0,C 180,E1 19697.311,E2 19697.311} C_VEL
LIN {X 0,Y 400.928,Z 491.78,A -85,B 0,C 180,E1 19694.969,E2 19694.969} C_VEL
LIN {X 0,Y 401.66,Z 480.988,A -85,B 0,C 180,E1 19692.77,E2 19692.77} C_VEL
LIN {X 0,Y 402.78,Z 467.849,A -85,B 0,C 180,E1 19690.572,E2 19690.572} C_VEL
LIN {X 0,Y 404.111,Z 454.026,A -85,B 0,C 180,E1 19688.673,E2 19688.673} C_VEL
LIN {X 0,Y 405.598,Z 439.256,A -85,B 0,C 180,E1 19687.002,E2 19687.002} C_VEL
LIN {X 0,Y 407.146,Z 423.63,A -85,B 0,C 180,E1 19685.558,E2 19685.558} C_VEL
LIN {X 0,Y 408.732,Z 406.448,A -85,B 0,C 180,E1 19684.288,E2 19684.288} C_VEL
LIN {X 0,Y 410.117,Z 389.231,A -85,B 0,C 180,E1 19683.309,E2 19683.309} C_VEL
LIN {X 0,Y 411.341,Z 370.743,A -85,B 0,C 180,E1 19682.547,E2 19682.547} C_VEL
LIN {X 0,Y 412.121,Z 352.232,A -85,B 0,C 180,E1 19682.046,E2 19682.046} C_VEL
LIN {X 0,Y 414.961,Z 170.981,A -85,B 0,C 180,E1 19678.906,E2 19678.906} C_VEL
LIN {X 0,Y 414.325,Z 156.312,A -85,B 0,C 180,E1 19678.545,E2 19678.545} C_VEL
LIN {X 0,Y 417.427,Z 111.483,A -85,B 0,C 180,E1 19675.862,E2 19675.862} C_VEL
LIN {X 0,Y 407.968,Z 87.55,A -85,B 0,C 180,E1 19673.501,E2 19673.501} C_VEL
LIN {X 0,Y 401.585,Z 72.301,A -85,B 0,C 180,E1 19671.827,E2 19671.827} C_VEL
LIN {X 0,Y 401.497,Z 71.784,A -85,B 0,C 180,E1 19671.497,E2 19671.497} C_VEL
LIN {X 0,Y 401.495,Z 71.786,A -85,B 0,C 180,E1 19667.488,E2 19667.488} C_VEL
LIN {X 0,Y 401.492,Z 71.783,A -85,B 0,C 180,E1 19663.559,E2 19663.559} C_VEL
LIN {X 0,Y 401.491,Z 71.787,A -85,B 0,C 180,E1 19659.608,E2 19659.608} C_VEL
LIN {X 0,Y 401.489,Z 71.78,A -85,B 0,C 180,E1 19655.644,E2 19655.644} C_VEL
LIN {X 0,Y 401.488,Z 71.78,A -85,B 0,C 180,E1 19651.7,E2 19651.7} C_VEL
LIN {X 0,Y 401.485,Z 71.779,A -85,B 0,C 180,E1 19647.756,E2 19647.756} C_VEL
LIN {X 0,Y 401.483,Z 71.776,A -85,B 0,C 180,E1 19643.794,E2 19643.794} C_VEL
LIN {X 0,Y 401.48,Z 71.779,A -85,B 0,C 180,E1 19639.797,E2 19639.797} C_VEL
LIN {X 0,Y 401.48,Z 71.784,A -85,B 0,C 180,E1 19635.899,E2 19635.899} C_VEL
LIN {X 0,Y 401.48,Z 71.786,A -85,B 0,C 180,E1 19631.929,E2 19631.929} C_VEL
LIN {X 0,Y 401.478,Z 71.784,A -85,B 0,C 180,E1 19628.017,E2 19628.017} C_VEL
LIN {X 0,Y 401.476,Z 71.779,A -85,B 0,C 180,E1 19623.998,E2 19623.998} C_VEL
LIN {X 0,Y 401.474,Z 71.775,A -85,B 0,C 180,E1 19620.142,E2 19620.142} C_VEL
LIN {X 0,Y 401.474,Z 71.782,A -85,B 0,C 180,E1 19616.144,E2 19616.144} C_VEL
LIN {X 0,Y 401.471,Z 71.786,A -85,B 0,C 180,E1 19612.271,E2 19612.271} C_VEL
LIN {X 0,Y 401.469,Z 71.787,A -85,B 0,C 180,E1 19608.361,E2 19608.361} C_VEL
LIN {X 0,Y 401.468,Z 71.786,A -85,B 0,C 180,E1 19604.396,E2 19604.396} C_VEL
LIN {X 0,Y 401.469,Z 71.786,A -85,B 0,C 180,E1 19600.504,E2 19600.504} C_VEL
LIN {X 0,Y 401.465,Z 71.755,A -85,B 0,C 180,E1 19596.516,E2 19596.516} C_VEL
LIN {X 0,Y 401.465,Z 71.788,A -85,B 0,C 180,E1 19592.564,E2 19592.564} C_VEL
LIN {X 0,Y 401.463,Z 71.776,A -85,B 0,C 180,E1 19588.632,E2 19588.632} C_VEL
LIN {X 0,Y 401.461,Z 71.772,A -85,B 0,C 180,E1 19584.703,E2 19584.703} C_VEL
LIN {X 0,Y 401.456,Z 71.789,A -85,B 0,C 180,E1 19580.941,E2 19580.941} C_VEL
LIN {X 0,Y 401.457,Z 71.786,A -85,B 0,C 180,E1 19576.967,E2 19576.967} C_VEL
LIN {X 0,Y 401.456,Z 71.781,A -85,B 0,C 180,E1 19573.031,E2 19573.031} C_VEL
LIN {X 0,Y 401.49,Z 72.034,A -85,B 0,C 180,E1 19570.873,E2 19570.873} C_VEL
LIN {X 0,Y 407.192,Z 89.543,A -85,B 0,C 180,E1 19568.322,E2 19568.322} C_VEL
LIN {X 0,Y 410.588,Z 102.744,A -85,B 0,C 180,E1 19566.523,E2 19566.523} C_VEL
LIN {X 0,Y 409.893,Z 136.321,A -85,B 0,C 180,E1 19562.693,E2 19562.693} C_VEL
LIN {X 0,Y 409.158,Z 171.065,A -85,B 0,C 180,E1 19558.776,E2 19558.776} C_VEL
LIN {X 0,Y 408.895,Z 196.757,A -85,B 0,C 180,E1 19556.01,E2 19556.01} C_VEL
LIN {X 0,Y 409.456,Z 201.816,A -85,B 0,C 180,E1 19555.881,E2 19555.881} C_VEL
LIN {X 0,Y 408.076,Z 306.143,A -85,B 0,C 180,E1 19554.006,E2 19554.006} C_VEL
LIN {X 0,Y 407.977,Z 321.963,A -85,B 0,C 180,E1 19553.491,E2 19553.491} C_VEL
LIN {X 0,Y 407.535,Z 336.921,A -85,B 0,C 180,E1 19552.706,E2 19552.706} C_VEL
LIN {X 0,Y 406.847,Z 350.226,A -85,B 0,C 180,E1 19551.725,E2 19551.725} C_VEL
LIN {X 0,Y 406.03,Z 362.412,A -85,B 0,C 180,E1 19550.541,E2 19550.541} C_VEL
LIN {X 0,Y 405.151,Z 373.507,A -85,B 0,C 180,E1 19549.16,E2 19549.16} C_VEL
LIN {X 0,Y 404.212,Z 383.508,A -85,B 0,C 180,E1 19547.563,E2 19547.563} C_VEL
LIN {X 0,Y 403.353,Z 392.018,A -85,B 0,C 180,E1 19545.822,E2 19545.822} C_VEL
LIN {X 0,Y 402.623,Z 399.072,A -85,B 0,C 180,E1 19543.937,E2 19543.937} C_VEL
LIN {X 0,Y 402.497,Z 400.23,A -85,B 0,C 180,E1 19543.557,E2 19543.557} C_VEL
LIN {X 0,Y 401.215,Z 403.229,A -85,B 0,C 180,E1 19542.551,E2 19542.551} C_VEL
LIN {X 0,Y 396.752,Z 407.541,A -85,B 0,C 180,E1 19540.838,E2 19540.838} C_VEL
LIN {X 0,Y 394.014,Z 409.895,A -85,B 0,C 180,E1 19539.478,E2 19539.478} C_VEL
LIN {X 0,Y 393.597,Z 410.597,A -85,B 0,C 180,E1 19538.844,E2 19538.844} C_VEL
LIN {X 0,Y 393.415,Z 411.689,A -85,B 0,C 180,E1 19536.566,E2 19536.566} C_VEL
LIN {X 0,Y 393.399,Z 410.94,A -85,B 0,C 180,E1 19534.372,E2 19534.372} C_VEL
LIN {X 0,Y 393.539,Z 408.42,A -85,B 0,C 180,E1 19532.183,E2 19532.183} C_VEL
LIN {X 0,Y 393.852,Z 403.999,A -85,B 0,C 180,E1 19529.999,E2 19529.999} C_VEL
LIN {X 0,Y 394.357,Z 397.422,A -85,B 0,C 180,E1 19527.819,E2 19527.819} C_VEL
LIN {X 0,Y 394.977,Z 389.65,A -85,B 0,C 180,E1 19525.934,E2 19525.934} C_VEL
LIN {X 0,Y 395.647,Z 381.24,A -85,B 0,C 180,E1 19524.343,E2 19524.343} C_VEL
LIN {X 0,Y 396.436,Z 370.575,A -85,B 0,C 180,E1 19522.754,E2 19522.754} C_VEL
LIN {X 0,Y 397.208,Z 358.053,A -85,B 0,C 180,E1 19521.312,E2 19521.312} C_VEL
LIN {X 0,Y 397.841,Z 345.807,A -85,B 0,C 180,E1 19520.232,E2 19520.232} C_VEL
LIN {X 0,Y 398.353,Z 332.248,A -85,B 0,C 180,E1 19519.331,E2 19519.331} C_VEL
LIN {X 0,Y 398.592,Z 316.896,A -85,B 0,C 180,E1 19518.629,E2 19518.629} C_VEL
LIN {X 0,Y 398.555,Z 300.282,A -85,B 0,C 180,E1 19518.201,E2 19518.201} C_VEL
LIN {X 0,Y 400.022,Z 193.414,A -85,B 0,C 180,E1 19516.263,E2 19516.263} C_VEL
LIN {X 0,Y 400.516,Z 183.164,A -85,B 0,C 180,E1 19515.609,E2 19515.609} C_VEL
LIN {X 0,Y 401.048,Z 154.122,A -85,B 0,C 180,E1 19513.636,E2 19513.636} C_VEL
LIN {X 0,Y 401.572,Z 153.003,A -85,B 0,C 180,E1 19513.398,E2 19513.398} C_VEL
LIN {X 0,Y 403.173,Z 153.686,A -85,B 0,C 180,E1 19513.132,E2 19513.132} C_VEL
LIN {X 0,Y 402.188,Z 170.142,A -85,B 0,C 180,E1 19511.744,E2 19511.744} C_VEL
LIN {X 0,Y 404.13,Z 194.014,A -85,B 0,C 180,E1 19511.099,E2 19511.099} C_VEL
LIN {X 0,Y 401.584,Z 298.945,A -85,B 0,C 180,E1 19508.942,E2 19508.942} C_VEL
LIN {X 0,Y 401.054,Z 315.006,A -85,B 0,C 180,E1 19508.347,E2 19508.347} C_VEL
LIN {X 0,Y 400.287,Z 329.879,A -85,B 0,C 180,E1 19507.531,E2 19507.531} C_VEL
LIN {X 0,Y 399.402,Z 343.409,A -85,B 0,C 180,E1 19506.544,E2 19506.544} C_VEL
LIN {X 0,Y 398.281,Z 357.376,A -85,B 0,C 180,E1 19505.212,E2 19505.212} C_VEL
LIN {X 0,Y 397.263,Z 369.148,A -85,B 0,C 180,E1 19503.786,E2 19503.786} C_VEL
LIN {X 0,Y 396.185,Z 380.552,A -85,B 0,C 180,E1 19502.044,E2 19502.044} C_VEL
LIN {X 0,Y 395.259,Z 390.015,A -85,B 0,C 180,E1 19500.189,E2 19500.189} C_VEL
LIN {X 0,Y 394.568,Z 397.364,A -85,B 0,C 180,E1 19498.361,E2 19498.361} C_VEL
LIN {X 0,Y 393.998,Z 403.742,A -85,B 0,C 180,E1 19496.236,E2 19496.236} C_VEL
LIN {X 0,Y 393.644,Z 408.307,A -85,B 0,C 180,E1 19494.073,E2 19494.073} C_VEL
LIN {X 0,Y 393.462,Z 411.25,A -85,B 0,C 180,E1 19491.68,E2 19491.68} C_VEL
LIN {X 0,Y 393.47,Z 412.103,A -85,B 0,C 180,E1 19489.418,E2 19489.418} C_VEL
LIN {X 0,Y 393.651,Z 411.253,A -85,B 0,C 180,E1 19487.228,E2 19487.228} C_VEL
LIN {X 0,Y 394.036,Z 408.428,A -85,B 0,C 180,E1 19484.931,E2 19484.931} C_VEL
LIN {X 0,Y 394.62,Z 403.942,A -85,B 0,C 180,E1 19482.769,E2 19482.769} C_VEL
LIN {X 0,Y 395.504,Z 397.104,A -85,B 0,C 180,E1 19480.52,E2 19480.52} C_VEL
LIN {X 0,Y 396.525,Z 389.122,A -85,B 0,C 180,E1 19478.585,E2 19478.585} C_VEL
LIN {X 0,Y 397.753,Z 379.396,A -85,B 0,C 180,E1 19476.747,E2 19476.747} C_VEL
LIN {X 0,Y 399.138,Z 367.48,A -85,B 0,C 180,E1 19475,E2 19475} C_VEL
LIN {X 0,Y 400.447,Z 355.06,A -85,B 0,C 180,E1 19473.575,E2 19473.575} C_VEL
LIN {X 0,Y 401.684,Z 341.562,A -85,B 0,C 180,E1 19472.356,E2 19472.356} C_VEL
LIN {X 0,Y 402.812,Z 325.979,A -85,B 0,C 180,E1 19471.298,E2 19471.298} C_VEL
LIN {X 0,Y 403.618,Z 310.62,A -85,B 0,C 180,E1 19470.551,E2 19470.551} C_VEL
LIN {X 0,Y 404.156,Z 294.21,A -85,B 0,C 180,E1 19470.033,E2 19470.033} C_VEL
LIN {X 0,Y 407.071,Z 202.514,A -85,B 0,C 180,E1 19467.99,E2 19467.99} C_VEL
LIN {X 0,Y 401.797,Z 173.824,A -85,B 0,C 180,E1 19466.84,E2 19466.84} C_VEL
LIN {X 0,Y 401.8,Z 171.677,A -85,B 0,C 180,E1 19466.611,E2 19466.611} C_VEL
LIN {X 0,Y 404.747,Z 144.527,A -85,B 0,C 180,E1 19462.496,E2 19462.496} C_VEL
LIN {X 0,Y 407.96,Z 118.486,A -85,B 0,C 180,E1 19458.482,E2 19458.482} C_VEL
LIN {X 0,Y 404.199,Z 103.928,A -85,B 0,C 180,E1 19455.496,E2 19455.496} C_VEL
LIN {X 0,Y 400.149,Z 90.973,A -85,B 0,C 180,E1 19452.556,E2 19452.556} C_VEL
LIN {X 0,Y 396.186,Z 79.733,A -85,B 0,C 180,E1 19449.735,E2 19449.735} C_VEL
LIN {X 0,Y 393.558,Z 72.909,A -85,B 0,C 180,E1 19447.805,E2 19447.805} C_VEL
LIN {X 0,Y 393.541,Z 72.777,A -85,B 0,C 180,E1 19443.934,E2 19443.934} C_VEL
LIN {X 0,Y 393.538,Z 72.777,A -85,B 0,C 180,E1 19440,E2 19440} C_VEL
LIN {X 0,Y 393.534,Z 72.776,A -85,B 0,C 180,E1 19436.067,E2 19436.067} C_VEL
LIN {X 0,Y 393.53,Z 72.776,A -85,B 0,C 180,E1 19432.114,E2 19432.114} C_VEL
LIN {X 0,Y 393.533,Z 72.775,A -85,B 0,C 180,E1 19428.273,E2 19428.273} C_VEL
LIN {X 0,Y 393.534,Z 72.776,A -85,B 0,C 180,E1 19424.352,E2 19424.352} C_VEL
LIN {X 0,Y 393.533,Z 72.778,A -85,B 0,C 180,E1 19420.405,E2 19420.405} C_VEL
LIN {X 0,Y 393.529,Z 72.78,A -85,B 0,C 180,E1 19416.491,E2 19416.491} C_VEL
LIN {X 0,Y 393.53,Z 72.777,A -85,B 0,C 180,E1 19412.621,E2 19412.621} C_VEL
LIN {X 0,Y 393.535,Z 72.776,A -85,B 0,C 180,E1 19408.782,E2 19408.782} C_VEL
LIN {X 0,Y 393.524,Z 72.782,A -85,B 0,C 180,E1 19404.777,E2 19404.777} C_VEL
LIN {X 0,Y 393.519,Z 72.779,A -85,B 0,C 180,E1 19400.801,E2 19400.801} C_VEL
LIN {X 0,Y 393.517,Z 72.779,A -85,B 0,C 180,E1 19396.884,E2 19396.884} C_VEL
LIN {X 0,Y 393.556,Z 73.177,A -85,B 0,C 180,E1 19396.161,E2 19396.161} C_VEL
LIN {X 0,Y 398.492,Z 84.681,A -85,B 0,C 180,E1 19393.433,E2 19393.433} C_VEL
LIN {X 0,Y 403.943,Z 98.476,A -85,B 0,C 180,E1 19390.617,E2 19390.617} C_VEL
LIN {X 0,Y 409.272,Z 113.777,A -85,B 0,C 180,E1 19387.899,E2 19387.899} C_VEL
LIN {X 0,Y 411.634,Z 121.968,A -85,B 0,C 180,E1 19386.607,E2 19386.607} C_VEL
LIN {X 0,Y 406.342,Z 161.535,A -85,B 0,C 180,E1 19382.347,E2 19382.347} C_VEL
LIN {X 0,Y 408.843,Z 184.707,A -85,B 0,C 180,E1 19381.662,E2 19381.662} C_VEL
LIN {X 0,Y 405.829,Z 343.937,A -85,B 0,C 180,E1 19378.838,E2 19378.838} C_VEL
LIN {X 0,Y 405.151,Z 362.809,A -85,B 0,C 180,E1 19378.395,E2 19378.395} C_VEL
LIN {X 0,Y 403.939,Z 380.623,A -85,B 0,C 180,E1 19377.734,E2 19377.734} C_VEL
LIN {X 0,Y 402.518,Z 397.146,A -85,B 0,C 180,E1 19376.879,E2 19376.879} C_VEL
LIN {X 0,Y 400.828,Z 414.138,A -85,B 0,C 180,E1 19375.725,E2 19375.725} C_VEL
LIN {X 0,Y 399.07,Z 430.27,A -85,B 0,C 180,E1 19374.341,E2 19374.341} C_VEL
LIN {X 0,Y 397.271,Z 446.186,A -85,B 0,C 180,E1 19372.649,E2 19372.649} C_VEL
LIN {X 0,Y 395.678,Z 460.581,A -85,B 0,C 180,E1 19370.777,E2 19370.777} C_VEL
LIN {X 0,Y 394.392,Z 473.266,A -85,B 0,C 180,E1 19368.783,E2 19368.783} C_VEL
LIN {X 0,Y 393.365,Z 485.097,A -85,B 0,C 180,E1 19366.541,E2 19366.541} C_VEL
LIN {X 0,Y 392.713,Z 495.801,A -85,B 0,C 180,E1 19364.062,E2 19364.062} C_VEL
LIN {X 0,Y 392.438,Z 504.736,A -85,B 0,C 180,E1 19361.464,E2 19361.464} C_VEL
LIN {X 0,Y 392.486,Z 511.517,A -85,B 0,C 180,E1 19358.941,E2 19358.941} C_VEL
LIN {X 0,Y 392.7,Z 516.541,A -85,B 0,C 180,E1 19356.433,E2 19356.433} C_VEL
LIN {X 0,Y 392.943,Z 519.907,A -85,B 0,C 180,E1 19353.941,E2 19353.941} C_VEL
LIN {X 0,Y 393.113,Z 521.669,A -85,B 0,C 180,E1 19351.459,E2 19351.459} C_VEL
LIN {X 0,Y 393.131,Z 521.823,A -85,B 0,C 180,E1 19348.981,E2 19348.981} C_VEL
LIN {X 0,Y 392.974,Z 520.385,A -85,B 0,C 180,E1 19346.5,E2 19346.5} C_VEL
LIN {X 0,Y 392.732,Z 517.34,A -85,B 0,C 180,E1 19344.01,E2 19344.01} C_VEL
LIN {X 0,Y 392.516,Z 512.627,A -85,B 0,C 180,E1 19341.505,E2 19341.505} C_VEL
LIN {X 0,Y 392.432,Z 506.143,A -85,B 0,C 180,E1 19338.985,E2 19338.985} C_VEL
LIN {X 0,Y 392.644,Z 497.73,A -85,B 0,C 180,E1 19336.452,E2 19336.452} C_VEL
LIN {X 0,Y 393.197,Z 487.46,A -85,B 0,C 180,E1 19333.99,E2 19333.99} C_VEL
LIN {X 0,Y 394.076,Z 476.334,A -85,B 0,C 180,E1 19331.817,E2 19331.817} C_VEL
LIN {X 0,Y 395.296,Z 463.345,A -85,B 0,C 180,E1 19329.727,E2 19329.727} C_VEL
LIN {X 0,Y 396.743,Z 449.354,A -85,B 0,C 180,E1 19327.868,E2 19327.868} C_VEL
LIN {X 0,Y 398.318,Z 434.47,A -85,B 0,C 180,E1 19326.243,E2 19326.243} C_VEL
LIN {X 0,Y 400.001,Z 417.861,A -85,B 0,C 180,E1 19324.776,E2 19324.776} C_VEL
LIN {X 0,Y 401.558,Z 401.233,A -85,B 0,C 180,E1 19323.613,E2 19323.613} C_VEL
LIN {X 0,Y 402.972,Z 383.749,A -85,B 0,C 180,E1 19322.678,E2 19322.678} C_VEL
LIN {X 0,Y 404.127,Z 365.576,A -85,B 0,C 180,E1 19321.982,E2 19321.982} C_VEL
LIN {X 0,Y 404.79,Z 346.971,A -85,B 0,C 180,E1 19321.53,E2 19321.53} C_VEL
LIN {X 0,Y 407.779,Z 173.044,A -85,B 0,C 180,E1 19318.476,E2 19318.476} C_VEL
LIN {X 0,Y 407.045,Z 156.734,A -85,B 0,C 180,E1 19318.082,E2 19318.082} C_VEL
LIN {X 0,Y 410.178,Z 114.013,A -85,B 0,C 180,E1 19315.479,E2 19315.479} C_VEL
LIN {X 0,Y 400.543,Z 89.631,A -85,B 0,C 180,E1 19313.016,E2 19313.016} C_VEL
LIN {X 0,Y 393.646,Z 73.351,A -85,B 0,C 180,E1 19311.174,E2 19311.174} C_VEL
LIN {X 0,Y 393.562,Z 72.801,A -85,B 0,C 180,E1 19310.948,E2 19310.948} C_VEL
LIN {X 0,Y 393.559,Z 72.776,A -85,B 0,C 180,E1 19306.892,E2 19306.892} C_VEL
LIN {X 0,Y 393.559,Z 72.773,A -85,B 0,C 180,E1 19302.911,E2 19302.911} C_VEL
LIN {X 0,Y 393.561,Z 72.772,A -85,B 0,C 180,E1 19298.979,E2 19298.979} C_VEL
LIN {X 0,Y 393.559,Z 72.766,A -85,B 0,C 180,E1 19295.041,E2 19295.041} C_VEL
LIN {X 0,Y 393.561,Z 72.768,A -85,B 0,C 180,E1 19291.046,E2 19291.046} C_VEL
LIN {X 0,Y 393.561,Z 72.767,A -85,B 0,C 180,E1 19287.049,E2 19287.049} C_VEL
LIN {X 0,Y 393.565,Z 72.762,A -85,B 0,C 180,E1 19283.031,E2 19283.031} C_VEL
LIN {X 0,Y 393.565,Z 72.763,A -85,B 0,C 180,E1 19278.977,E2 19278.977} C_VEL
LIN {X 0,Y 393.569,Z 72.767,A -85,B 0,C 180,E1 19275.018,E2 19275.018} C_VEL
LIN {X 0,Y 393.564,Z 72.773,A -85,B 0,C 180,E1 19270.984,E2 19270.984} C_VEL
LIN {X 0,Y 393.569,Z 72.773,A -85,B 0,C 180,E1 19267.004,E2 19267.004} C_VEL
LIN {X 0,Y 393.559,Z 72.771,A -85,B 0,C 180,E1 19262.912,E2 19262.912} C_VEL
LIN {X 0,Y 393.56,Z 72.765,A -85,B 0,C 180,E1 19258.981,E2 19258.981} C_VEL
LIN {X 0,Y 393.556,Z 72.765,A -85,B 0,C 180,E1 19255.044,E2 19255.044} C_VEL
LIN {X 0,Y 393.554,Z 72.767,A -85,B 0,C 180,E1 19251.084,E2 19251.084} C_VEL
LIN {X 0,Y 393.549,Z 72.769,A -85,B 0,C 180,E1 19247.081,E2 19247.081} C_VEL
LIN {X 0,Y 393.549,Z 72.772,A -85,B 0,C 180,E1 19243.164,E2 19243.164} C_VEL
LIN {X 0,Y 393.543,Z 72.772,A -85,B 0,C 180,E1 19239.164,E2 19239.164} C_VEL
LIN {X 0,Y 393.547,Z 72.747,A -85,B 0,C 180,E1 19235.375,E2 19235.375} C_VEL
LIN {X 0,Y 393.548,Z 72.765,A -85,B 0,C 180,E1 19231.468,E2 19231.468} C_VEL
LIN {X 0,Y 393.549,Z 72.774,A -85,B 0,C 180,E1 19227.583,E2 19227.583} C_VEL
LIN {X 0,Y 393.544,Z 72.76,A -85,B 0,C 180,E1 19223.644,E2 19223.644} C_VEL
LIN {X 0,Y 393.551,Z 72.761,A -85,B 0,C 180,E1 19219.81,E2 19219.81} C_VEL
LIN {X 0,Y 393.545,Z 72.764,A -85,B 0,C 180,E1 19215.881,E2 19215.881} C_VEL
LIN {X 0,Y 393.545,Z 72.776,A -85,B 0,C 180,E1 19211.891,E2 19211.891} C_VEL
LIN {X 0,Y 393.574,Z 73.168,A -85,B 0,C 180,E1 19211.458,E2 19211.458} C_VEL
LIN {X 0,Y 399.591,Z 91.184,A -85,B 0,C 180,E1 19208.79,E2 19208.79} C_VEL
LIN {X 0,Y 403.3,Z 104.999,A -85,B 0,C 180,E1 19206.865,E2 19206.865} C_VEL
LIN {X 0,Y 402.545,Z 139.141,A -85,B 0,C 180,E1 19202.952,E2 19202.952} C_VEL
LIN {X 0,Y 401.749,Z 174.511,A -85,B 0,C 180,E1 19198.949,E2 19198.949} C_VEL
LIN {X 0,Y 401.5,Z 197.839,A -85,B 0,C 180,E1 19196.435,E2 19196.435} C_VEL
LIN {X 0,Y 402.07,Z 202.84,A -85,B 0,C 180,E1 19196.304,E2 19196.304} C_VEL
LIN {X 0,Y 400.612,Z 306.488,A -85,B 0,C 180,E1 19194.411,E2 19194.411} C_VEL
LIN {X 0,Y 400.521,Z 321.783,A -85,B 0,C 180,E1 19193.921,E2 19193.921} C_VEL
LIN {X 0,Y 400.12,Z 335.728,A -85,B 0,C 180,E1 19193.211,E2 19193.211} C_VEL
LIN {X 0,Y 399.468,Z 348.848,A -85,B 0,C 180,E1 19192.283,E2 19192.283} C_VEL
LIN {X 0,Y 398.551,Z 362.13,A -85,B 0,C 180,E1 19191.022,E2 19191.022} C_VEL
LIN {X 0,Y 397.558,Z 374.015,A -85,B 0,C 180,E1 19189.54,E2 19189.54} C_VEL
LIN {X 0,Y 396.554,Z 384.158,A -85,B 0,C 180,E1 19187.914,E2 19187.914} C_VEL
LIN {X 0,Y 395.63,Z 392.78,A -85,B 0,C 180,E1 19186.139,E2 19186.139} C_VEL
LIN {X 0,Y 394.837,Z 399.913,A -85,B 0,C 180,E1 19184.218,E2 19184.218} C_VEL
LIN {X 0,Y 394.202,Z 405.457,A -85,B 0,C 180,E1 19182.152,E2 19182.152} C_VEL
LIN {X 0,Y 393.77,Z 409.158,A -85,B 0,C 180,E1 19180.089,E2 19180.089} C_VEL
LIN {X 0,Y 393.597,Z 410.597,A -85,B 0,C 180,E1 19178.844,E2 19178.844} C_VEL
LIN {X 0,Y 392.522,Z 411.611,A -85,B 0,C 180,E1 19177.731,E2 19177.731} C_VEL
LIN {X 0,Y 388.547,Z 412.466,A -85,B 0,C 180,E1 19175.937,E2 19175.937} C_VEL
LIN {X 0,Y 385.914,Z 412.126,A -85,B 0,C 180,E1 19174.498,E2 19174.498} C_VEL
LIN {X 0,Y 385.494,Z 411.524,A -85,B 0,C 180,E1 19173.761,E2 19173.761} C_VEL
LIN {X 0,Y 385.697,Z 408.412,A -85,B 0,C 180,E1 19171.484,E2 19171.484} C_VEL
LIN {X 0,Y 386.08,Z 403.363,A -85,B 0,C 180,E1 19169.257,E2 19169.257} C_VEL
LIN {X 0,Y 386.631,Z 396.629,A -85,B 0,C 180,E1 19167.183,E2 19167.183} C_VEL
LIN {X 0,Y 387.277,Z 389.026,A -85,B 0,C 180,E1 19165.408,E2 19165.408} C_VEL
LIN {X 0,Y 388.081,Z 379.257,A -85,B 0,C 180,E1 19163.638,E2 19163.638} C_VEL
LIN {X 0,Y 388.942,Z 367.685,A -85,B 0,C 180,E1 19162.02,E2 19162.02} C_VEL
LIN {X 0,Y 389.681,Z 355.442,A -85,B 0,C 180,E1 19160.696,E2 19160.696} C_VEL
LIN {X 0,Y 390.313,Z 343.076,A -85,B 0,C 180,E1 19159.669,E2 19159.669} C_VEL
LIN {X 0,Y 390.788,Z 328.639,A -85,B 0,C 180,E1 19158.786,E2 19158.786} C_VEL
LIN {X 0,Y 390.949,Z 312.944,A -85,B 0,C 180,E1 19158.157,E2 19158.157} C_VEL
LIN {X 0,Y 390.986,Z 282.845,A -85,B 0,C 180,E1 19157.543,E2 19157.543} C_VEL
LIN {X 0,Y 392.416,Z 194.515,A -85,B 0,C 180,E1 19155.916,E2 19155.916} C_VEL
LIN {X 0,Y 392.965,Z 185.484,A -85,B 0,C 180,E1 19155.334,E2 19155.334} C_VEL
LIN {X 0,Y 393.424,Z 160.117,A -85,B 0,C 180,E1 19153.614,E2 19153.614} C_VEL
LIN {X 0,Y 393.947,Z 158.988,A -85,B 0,C 180,E1 19153.371,E2 19153.371} C_VEL
LIN {X 0,Y 395.425,Z 159.808,A -85,B 0,C 180,E1 19153.094,E2 19153.094} C_VEL
LIN {X 0,Y 394.79,Z 169.473,A -85,B 0,C 180,E1 19152.26,E2 19152.26} C_VEL
LIN {X 0,Y 396.794,Z 194.714,A -85,B 0,C 180,E1 19151.549,E2 19151.549} C_VEL
LIN {X 0,Y 394.113,Z 299.594,A -85,B 0,C 180,E1 19149.345,E2 19149.345} C_VEL
LIN {X 0,Y 393.561,Z 315.52,A -85,B 0,C 180,E1 19148.744,E2 19148.744} C_VEL
LIN {X 0,Y 392.762,Z 330.368,A -85,B 0,C 180,E1 19147.918,E2 19147.918} C_VEL
LIN {X 0,Y 391.781,Z 344.617,A -85,B 0,C 180,E1 19146.857,E2 19146.857} C_VEL
LIN {X 0,Y 390.61,Z 358.514,A -85,B 0,C 180,E1 19145.5,E2 19145.5} C_VEL
LIN {X 0,Y 389.524,Z 370.389,A -85,B 0,C 180,E1 19144.024,E2 19144.024} C_VEL
LIN {X 0,Y 388.434,Z 381.383,A -85,B 0,C 180,E1 19142.312,E2 19142.312} C_VEL
LIN {X 0,Y 387.454,Z 390.896,A -85,B 0,C 180,E1 19140.42,E2 19140.42} C_VEL
LIN {X 0,Y 386.707,Z 398.43,A -85,B 0,C 180,E1 19138.514,E2 19138.514} C_VEL
LIN {X 0,Y 386.105,Z 404.818,A -85,B 0,C 180,E1 19136.345,E2 19136.345} C_VEL
LIN {X 0,Y 385.73,Z 409.39,A -85,B 0,C 180,E1 19134.138,E2 19134.138} C_VEL
LIN {X 0,Y 385.539,Z 412.353,A -85,B 0,C 180,E1 19131.696,E2 19131.696} C_VEL
LIN {X 0,Y 385.551,Z 413.229,A -85,B 0,C 180,E1 19129.388,E2 19129.388} C_VEL
LIN {X 0,Y 385.743,Z 412.42,A -85,B 0,C 180,E1 19127.185,E2 19127.185} C_VEL
LIN {X 0,Y 386.123,Z 409.891,A -85,B 0,C 180,E1 19124.986,E2 19124.986} C_VEL
LIN {X 0,Y 386.739,Z 405.543,A -85,B 0,C 180,E1 19122.756,E2 19122.756} C_VEL
LIN {X 0,Y 387.564,Z 399.586,A -85,B 0,C 180,E1 19120.669,E2 19120.669} C_VEL
LIN {X 0,Y 388.608,Z 392.103,A -85,B 0,C 180,E1 19118.699,E2 19118.699} C_VEL
LIN {X 0,Y 389.832,Z 382.971,A -85,B 0,C 180,E1 19116.847,E2 19116.847} C_VEL
LIN {X 0,Y 391.229,Z 372.073,A -85,B 0,C 180,E1 19115.102,E2 19115.102} C_VEL
LIN {X 0,Y 392.659,Z 359.626,A -85,B 0,C 180,E1 19113.544,E2 19113.544} C_VEL
LIN {X 0,Y 393.987,Z 346.525,A -85,B 0,C 180,E1 19112.253,E2 19112.253} C_VEL
LIN {X 0,Y 395.249,Z 331.478,A -85,B 0,C 180,E1 19111.111,E2 19111.111} C_VEL
LIN {X 0,Y 396.243,Z 315.427,A -85,B 0,C 180,E1 19110.231,E2 19110.231} C_VEL
LIN {X 0,Y 396.886,Z 299.647,A -85,B 0,C 180,E1 19109.651,E2 19109.651} C_VEL
LIN {X 0,Y 400.089,Z 203.725,A -85,B 0,C 180,E1 19107.447,E2 19107.447} C_VEL
LIN {X 0,Y 394.868,Z 175.056,A -85,B 0,C 180,E1 19106.263,E2 19106.263} C_VEL
LIN {X 0,Y 394.51,Z 172.655,A -85,B 0,C 180,E1 19106.127,E2 19106.127} C_VEL
LIN {X 0,Y 397.712,Z 144.82,A -85,B 0,C 180,E1 19101.844,E2 19101.844} C_VEL
LIN {X 0,Y 400.792,Z 121.45,A -85,B 0,C 180,E1 19098.17,E2 19098.17} C_VEL
LIN {X 0,Y 397.165,Z 107.211,A -85,B 0,C 180,E1 19095.178,E2 19095.178} C_VEL
LIN {X 0,Y 393.002,Z 93.793,A -85,B 0,C 180,E1 19092.042,E2 19092.042} C_VEL
LIN {X 0,Y 389.199,Z 83.372,A -85,B 0,C 180,E1 19089.315,E2 19089.315} C_VEL
LIN {X 0,Y 386.587,Z 76.77,A -85,B 0,C 180,E1 19087.431,E2 19087.431} C_VEL
LIN {X 0,Y 385.623,Z 73.847,A -85,B 0,C 180,E1 19086.476,E2 19086.476} C_VEL
LIN {X 0,Y 385.614,Z 73.764,A -85,B 0,C 180,E1 19082.378,E2 19082.378} C_VEL
LIN {X 0,Y 385.616,Z 73.765,A -85,B 0,C 180,E1 19078.366,E2 19078.366} C_VEL
LIN {X 0,Y 385.611,Z 73.763,A -85,B 0,C 180,E1 19074.346,E2 19074.346} C_VEL
LIN {X 0,Y 385.61,Z 73.763,A -85,B 0,C 180,E1 19070.448,E2 19070.448} C_VEL
LIN {X 0,Y 385.608,Z 73.764,A -85,B 0,C 180,E1 19066.496,E2 19066.496} C_VEL
LIN {X 0,Y 385.6,Z 73.766,A -85,B 0,C 180,E1 19062.495,E2 19062.495} C_VEL
LIN {X 0,Y 385.598,Z 73.767,A -85,B 0,C 180,E1 19058.555,E2 19058.555} C_VEL
LIN {X 0,Y 385.597,Z 73.765,A -85,B 0,C 180,E1 19054.669,E2 19054.669} C_VEL
LIN {X 0,Y 385.587,Z 73.766,A -85,B 0,C 180,E1 19050.654,E2 19050.654} C_VEL
LIN {X 0,Y 385.592,Z 73.767,A -85,B 0,C 180,E1 19046.83,E2 19046.83} C_VEL
LIN {X 0,Y 385.579,Z 73.769,A -85,B 0,C 180,E1 19042.759,E2 19042.759} C_VEL
LIN {X 0,Y 385.591,Z 73.767,A -85,B 0,C 180,E1 19038.989,E2 19038.989} C_VEL
LIN {X 0,Y 385.631,Z 74.087,A -85,B 0,C 180,E1 19037.471,E2 19037.471} C_VEL
LIN {X 0,Y 390.759,Z 85.914,A -85,B 0,C 180,E1 19034.448,E2 19034.448} C_VEL
LIN {X 0,Y 395.998,Z 98.995,A -85,B 0,C 180,E1 19031.61,E2 19031.61} C_VEL
LIN {X 0,Y 401.192,Z 113.668,A -85,B 0,C 180,E1 19028.859,E2 19028.859} C_VEL
LIN {X 0,Y 404.515,Z 124.936,A -85,B 0,C 180,E1 19026.976,E2 19026.976} C_VEL
LIN {X 0,Y 399.311,Z 161.84,A -85,B 0,C 180,E1 19022.929,E2 19022.929} C_VEL
LIN {X 0,Y 401.874,Z 185.542,A -85,B 0,C 180,E1 19022.208,E2 19022.208} C_VEL
LIN {X 0,Y 398.339,Z 354.248,A -85,B 0,C 180,E1 19019.121,E2 19019.121} C_VEL
LIN {X 0,Y 397.253,Z 372.657,A -85,B 0,C 180,E1 19018.537,E2 19018.537} C_VEL
LIN {X 0,Y 395.745,Z 390.539,A -85,B 0,C 180,E1 19017.703,E2 19017.703} C_VEL
LIN {X 0,Y 394.003,Z 407.957,A -85,B 0,C 180,E1 19016.602,E2 19016.602} C_VEL
LIN {X 0,Y 392.174,Z 424.26,A -85,B 0,C 180,E1 19015.281,E2 19015.281} C_VEL
LIN {X 0,Y 390.321,Z 439.791,A -85,B 0,C 180,E1 19013.715,E2 19013.715} C_VEL
LIN {X 0,Y 388.565,Z 454.427,A -85,B 0,C 180,E1 19011.909,E2 19011.909} C_VEL
LIN {X 0,Y 387.035,Z 467.93,A -85,B 0,C 180,E1 19009.89,E2 19009.89} C_VEL
LIN {X 0,Y 385.806,Z 480.248,A -85,B 0,C 180,E1 19007.652,E2 19007.652} C_VEL
LIN {X 0,Y 384.949,Z 491.274,A -85,B 0,C 180,E1 19005.21,E2 19005.21} C_VEL
LIN {X 0,Y 384.537,Z 500.242,A -85,B 0,C 180,E1 19002.77,E2 19002.77} C_VEL
LIN {X 0,Y 384.449,Z 507.8,A -85,B 0,C 180,E1 19000.187,E2 19000.187} C_VEL
LIN {X 0,Y 384.641,Z 513.824,A -85,B 0,C 180,E1 18997.469,E2 18997.469} C_VEL
LIN {X 0,Y 384.926,Z 517.945,A -85,B 0,C 180,E1 18994.769,E2 18994.769} C_VEL
LIN {X 0,Y 385.148,Z 520.167,A -85,B 0,C 180,E1 18992.233,E2 18992.233} C_VEL
LIN {X 0,Y 385.224,Z 520.799,A -85,B 0,C 180,E1 18989.704,E2 18989.704} C_VEL
LIN {X 0,Y 385.101,Z 519.835,A -85,B 0,C 180,E1 18987.174,E2 18987.174} C_VEL
LIN {X 0,Y 384.859,Z 517.261,A -85,B 0,C 180,E1 18984.635,E2 18984.635} C_VEL
LIN {X 0,Y 384.596,Z 513.02,A -85,B 0,C 180,E1 18982.081,E2 18982.081} C_VEL
LIN {X 0,Y 384.45,Z 506.835,A -85,B 0,C 180,E1 18979.446,E2 18979.446} C_VEL
LIN {X 0,Y 384.584,Z 499.117,A -85,B 0,C 180,E1 18976.929,E2 18976.929} C_VEL
LIN {X 0,Y 385.059,Z 489.516,A -85,B 0,C 180,E1 18974.44,E2 18974.44} C_VEL
LIN {X 0,Y 385.95,Z 478.108,A -85,B 0,C 180,E1 18972.046,E2 18972.046} C_VEL
LIN {X 0,Y 387.142,Z 465.711,A -85,B 0,C 180,E1 18969.912,E2 18969.912} C_VEL
LIN {X 0,Y 388.636,Z 451.817,A -85,B 0,C 180,E1 18967.939,E2 18967.939} C_VEL
LIN {X 0,Y 390.288,Z 436.942,A -85,B 0,C 180,E1 18966.205,E2 18966.205} C_VEL
LIN {X 0,Y 391.998,Z 421.158,A -85,B 0,C 180,E1 18964.709,E2 18964.709} C_VEL
LIN {X 0,Y 393.683,Z 404.456,A -85,B 0,C 180,E1 18963.451,E2 18963.451} C_VEL
LIN {X 0,Y 395.215,Z 386.667,A -85,B 0,C 180,E1 18962.423,E2 18962.423} C_VEL
LIN {X 0,Y 396.496,Z 368.569,A -85,B 0,C 180,E1 18961.668,E2 18961.668} C_VEL
LIN {X 0,Y 397.305,Z 349.823,A -85,B 0,C 180,E1 18961.159,E2 18961.159} C_VEL
LIN {X 0,Y 400.483,Z 172.856,A -85,B 0,C 180,E1 18957.986,E2 18957.986} C_VEL
LIN {X 0,Y 399.78,Z 157.035,A -85,B 0,C 180,E1 18957.601,E2 18957.601} C_VEL
LIN {X 0,Y 402.937,Z 116.591,A -85,B 0,C 180,E1 18955.096,E2 18955.096} C_VEL
LIN {X 0,Y 393.479,Z 92.611,A -85,B 0,C 180,E1 18952.606,E2 18952.606} C_VEL
LIN {X 0,Y 385.719,Z 74.322,A -85,B 0,C 180,E1 18950.485,E2 18950.485} C_VEL
LIN {X 0,Y 385.625,Z 73.76,A -85,B 0,C 180,E1 18950.128,E2 18950.128} C_VEL
LIN {X 0,Y 385.623,Z 73.76,A -85,B 0,C 180,E1 18946.121,E2 18946.121} C_VEL
LIN {X 0,Y 385.625,Z 73.762,A -85,B 0,C 180,E1 18941.986,E2 18941.986} C_VEL
LIN {X 0,Y 385.62,Z 73.76,A -85,B 0,C 180,E1 18937.916,E2 18937.916} C_VEL
LIN {X 0,Y 385.616,Z 73.766,A -85,B 0,C 180,E1 18933.881,E2 18933.881} C_VEL
LIN {X 0,Y 385.613,Z 73.765,A -85,B 0,C 180,E1 18929.857,E2 18929.857} C_VEL
LIN {X 0,Y 385.609,Z 73.764,A -85,B 0,C 180,E1 18925.824,E2 18925.824} C_VEL
LIN {X 0,Y 385.607,Z 73.764,A -85,B 0,C 180,E1 18921.764,E2 18921.764} C_VEL
LIN {X 0,Y 385.603,Z 73.762,A -85,B 0,C 180,E1 18917.816,E2 18917.816} C_VEL
LIN {X 0,Y 385.602,Z 73.757,A -85,B 0,C 180,E1 18913.801,E2 18913.801} C_VEL
LIN {X 0,Y 385.601,Z 73.753,A -85,B 0,C 180,E1 18909.837,E2 18909.837} C_VEL
LIN {X 0,Y 385.6,Z 73.76,A -85,B 0,C 180,E1 18905.953,E2 18905.953} C_VEL
LIN {X 0,Y 385.602,Z 73.762,A -85,B 0,C 180,E1 18901.931,E2 18901.931} C_VEL
LIN {X 0,Y 385.602,Z 73.763,A -85,B 0,C 180,E1 18897.919,E2 18897.919} C_VEL
LIN {X 0,Y 385.604,Z 73.759,A -85,B 0,C 180,E1 18893.897,E2 18893.897} C_VEL
LIN {X 0,Y 385.601,Z 73.754,A -85,B 0,C 180,E1 18889.995,E2 18889.995} C_VEL
LIN {X 0,Y 385.601,Z 73.754,A -85,B 0,C 180,E1 18886.045,E2 18886.045} C_VEL
LIN {X 0,Y 385.604,Z 73.755,A -85,B 0,C 180,E1 18882.027,E2 18882.027} C_VEL
LIN {X 0,Y 385.605,Z 73.749,A -85,B 0,C 180,E1 18878.075,E2 18878.075} C_VEL
LIN {X 0,Y 385.612,Z 73.757,A -85,B 0,C 180,E1 18874.01,E2 18874.01} C_VEL
LIN {X 0,Y 385.606,Z 73.74,A -85,B 0,C 180,E1 18870.142,E2 18870.142} C_VEL
LIN {X 0,Y 385.614,Z 73.762,A -85,B 0,C 180,E1 18866.118,E2 18866.118} C_VEL
LIN {X 0,Y 385.623,Z 73.767,A -85,B 0,C 180,E1 18862.017,E2 18862.017} C_VEL
LIN {X 0,Y 385.619,Z 73.765,A -85,B 0,C 180,E1 18858.013,E2 18858.013} C_VEL
LIN {X 0,Y 385.613,Z 73.762,A -85,B 0,C 180,E1 18854.017,E2 18854.017} C_VEL
LIN {X 0,Y 385.64,Z 73.943,A -85,B 0,C 180,E1 18852.182,E2 18852.182} C_VEL
LIN {X 0,Y 387.005,Z 78.171,A -85,B 0,C 180,E1 18851.475,E2 18851.475} C_VEL
LIN {X 0,Y 392.384,Z 94.027,A -85,B 0,C 180,E1 18849.111,E2 18849.111} C_VEL
LIN {X 0,Y 396.055,Z 107.46,A -85,B 0,C 180,E1 18847.209,E2 18847.209} C_VEL
LIN {X 0,Y 395.22,Z 142.138,A -85,B 0,C 180,E1 18843.209,E2 18843.209} C_VEL
LIN {X 0,Y 394.383,Z 177.335,A -85,B 0,C 180,E1 18839.21,E2 18839.21} C_VEL
LIN {X 0,Y 394.113,Z 198.834,A -85,B 0,C 180,E1 18836.88,E2 18836.88} C_VEL
LIN {X 0,Y 394.707,Z 203.77,A -85,B 0,C 180,E1 18836.744,E2 18836.744} C_VEL
LIN {X 0,Y 393.168,Z 307.04,A -85,B 0,C 180,E1 18834.827,E2 18834.827} C_VEL
LIN {X 0,Y 393.086,Z 321.929,A -85,B 0,C 180,E1 18834.354,E2 18834.354} C_VEL
LIN {X 0,Y 392.677,Z 336.034,A -85,B 0,C 180,E1 18833.641,E2 18833.641} C_VEL
LIN {X 0,Y 391.958,Z 349.862,A -85,B 0,C 180,E1 18832.654,E2 18832.654} C_VEL
LIN {X 0,Y 390.987,Z 363.165,A -85,B 0,C 180,E1 18831.37,E2 18831.37} C_VEL
LIN {X 0,Y 389.933,Z 375.065,A -85,B 0,C 180,E1 18829.86,E2 18829.86} C_VEL
LIN {X 0,Y 388.912,Z 384.811,A -85,B 0,C 180,E1 18828.278,E2 18828.278} C_VEL
LIN {X 0,Y 387.921,Z 393.544,A -85,B 0,C 180,E1 18826.469,E2 18826.469} C_VEL
LIN {X 0,Y 387.005,Z 401.225,A -85,B 0,C 180,E1 18824.359,E2 18824.359} C_VEL
LIN {X 0,Y 386.293,Z 407.042,A -85,B 0,C 180,E1 18822.101,E2 18822.101} C_VEL
LIN {X 0,Y 385.819,Z 410.736,A -85,B 0,C 180,E1 18819.847,E2 18819.847} C_VEL
LIN {X 0,Y 385.552,Z 412.548,A -85,B 0,C 180,E1 18817.599,E2 18817.599} C_VEL
LIN {X 0,Y 385.461,Z 412.585,A -85,B 0,C 180,E1 18815.357,E2 18815.357} C_VEL
LIN {X 0,Y 385.494,Z 411.524,A -85,B 0,C 180,E1 18813.761,E2 18813.761} C_VEL
LIN {X 0,Y 384.575,Z 410.351,A -85,B 0,C 180,E1 18812.627,E2 18812.627} C_VEL
LIN {X 0,Y 380.581,Z 407.601,A -85,B 0,C 180,E1 18810.659,E2 18810.659} C_VEL
LIN {X 0,Y 378.491,Z 404.823,A -85,B 0,C 180,E1 18809.324,E2 18809.324} C_VEL
LIN {X 0,Y 378.286,Z 403.154,A -85,B 0,C 180,E1 18808.7,E2 18808.7} C_VEL
LIN {X 0,Y 378.888,Z 396.318,A -85,B 0,C 180,E1 18806.671,E2 18806.671} C_VEL
LIN {X 0,Y 379.668,Z 387.553,A -85,B 0,C 180,E1 18804.71,E2 18804.71} C_VEL
LIN {X 0,Y 380.554,Z 376.999,A -85,B 0,C 180,E1 18802.906,E2 18802.906} C_VEL
LIN {X 0,Y 381.389,Z 365.692,A -85,B 0,C 180,E1 18801.405,E2 18801.405} C_VEL
LIN {X 0,Y 382.1,Z 354.214,A -85,B 0,C 180,E1 18800.206,E2 18800.206} C_VEL
LIN {X 0,Y 382.805,Z 339.969,A -85,B 0,C 180,E1 18799.083,E2 18799.083} C_VEL
LIN {X 0,Y 383.212,Z 324.593,A -85,B 0,C 180,E1 18798.233,E2 18798.233} C_VEL
LIN {X 0,Y 383.282,Z 308.796,A -85,B 0,C 180,E1 18797.695,E2 18797.695} C_VEL
LIN {X 0,Y 384.257,Z 225.303,A -85,B 0,C 180,E1 18796.127,E2 18796.127} C_VEL
LIN {X 0,Y 384.825,Z 195.622,A -85,B 0,C 180,E1 18795.555,E2 18795.555} C_VEL
LIN {X 0,Y 385.435,Z 186.474,A -85,B 0,C 180,E1 18794.964,E2 18794.964} C_VEL
LIN {X 0,Y 385.853,Z 165.873,A -85,B 0,C 180,E1 18793.554,E2 18793.554} C_VEL
LIN {X 0,Y 386.429,Z 164.969,A -85,B 0,C 180,E1 18793.308,E2 18793.308} C_VEL
LIN {X 0,Y 387.669,Z 165.583,A -85,B 0,C 180,E1 18793.093,E2 18793.093} C_VEL
LIN {X 0,Y 387.469,Z 170.368,A -85,B 0,C 180,E1 18792.717,E2 18792.717} C_VEL
LIN {X 0,Y 389.476,Z 195.494,A -85,B 0,C 180,E1 18792.013,E2 18792.013} C_VEL
LIN {X 0,Y 386.664,Z 300.061,A -85,B 0,C 180,E1 18789.768,E2 18789.768} C_VEL
LIN {X 0,Y 386.075,Z 316.213,A -85,B 0,C 180,E1 18789.146,E2 18789.146} C_VEL
LIN {X 0,Y 385.19,Z 331.783,A -85,B 0,C 180,E1 18788.257,E2 18788.257} C_VEL
LIN {X 0,Y 384.125,Z 346.258,A -85,B 0,C 180,E1 18787.139,E2 18787.139} C_VEL
LIN {X 0,Y 382.948,Z 359.636,A -85,B 0,C 180,E1 18785.799,E2 18785.799} C_VEL
LIN {X 0,Y 381.761,Z 371.925,A -85,B 0,C 180,E1 18784.229,E2 18784.229} C_VEL
LIN {X 0,Y 380.611,Z 382.929,A -85,B 0,C 180,E1 18782.46,E2 18782.46} C_VEL
LIN {X 0,Y 379.534,Z 392.972,A -85,B 0,C 180,E1 18780.386,E2 18780.386} C_VEL
LIN {X 0,Y 378.72,Z 400.668,A -85,B 0,C 180,E1 18778.305,E2 18778.305} C_VEL
LIN {X 0,Y 378.136,Z 406.799,A -85,B 0,C 180,E1 18776.087,E2 18776.087} C_VEL
LIN {X 0,Y 377.766,Z 411.046,A -85,B 0,C 180,E1 18773.826,E2 18773.826} C_VEL
LIN {X 0,Y 377.608,Z 413.595,A -85,B 0,C 180,E1 18771.519,E2 18771.519} C_VEL
LIN {X 0,Y 377.656,Z 414.352,A -85,B 0,C 180,E1 18768.987,E2 18768.987} C_VEL
LIN {X 0,Y 377.899,Z 413.222,A -85,B 0,C 180,E1 18766.687,E2 18766.687} C_VEL
LIN {X 0,Y 378.399,Z 410.159,A -85,B 0,C 180,E1 18764.268,E2 18764.268} C_VEL
LIN {X 0,Y 379.139,Z 405.193,A -85,B 0,C 180,E1 18761.953,E2 18761.953} C_VEL
LIN {X 0,Y 380.116,Z 398.728,A -85,B 0,C 180,E1 18759.818,E2 18759.818} C_VEL
LIN {X 0,Y 381.423,Z 389.863,A -85,B 0,C 180,E1 18757.647,E2 18757.647} C_VEL
LIN {X 0,Y 382.795,Z 380.131,A -85,B 0,C 180,E1 18755.81,E2 18755.81} C_VEL
LIN {X 0,Y 384.286,Z 368.831,A -85,B 0,C 180,E1 18754.116,E2 18754.116} C_VEL
LIN {X 0,Y 385.793,Z 356.041,A -85,B 0,C 180,E1 18752.616,E2 18752.616} C_VEL
LIN {X 0,Y 387.135,Z 342.903,A -85,B 0,C 180,E1 18751.4,E2 18751.4} C_VEL
LIN {X 0,Y 388.411,Z 327.24,A -85,B 0,C 180,E1 18750.302,E2 18750.302} C_VEL
LIN {X 0,Y 389.325,Z 311.63,A -85,B 0,C 180,E1 18749.521,E2 18749.521} C_VEL
LIN {X 0,Y 389.926,Z 295.356,A -85,B 0,C 180,E1 18748.989,E2 18748.989} C_VEL
LIN {X 0,Y 393.158,Z 205.004,A -85,B 0,C 180,E1 18746.886,E2 18746.886} C_VEL
LIN {X 0,Y 388.065,Z 176.706,A -85,B 0,C 180,E1 18745.68,E2 18745.68} C_VEL
LIN {X 0,Y 387.357,Z 172.503,A -85,B 0,C 180,E1 18745.454,E2 18745.454} C_VEL
LIN {X 0,Y 390.755,Z 145.088,A -85,B 0,C 180,E1 18741.149,E2 18741.149} C_VEL
LIN {X 0,Y 393.598,Z 124.276,A -85,B 0,C 180,E1 18737.825,E2 18737.825} C_VEL
LIN {X 0,Y 390.319,Z 111.156,A -85,B 0,C 180,E1 18734.995,E2 18734.995} C_VEL
LIN {X 0,Y 386.259,Z 97.791,A -85,B 0,C 180,E1 18731.8,E2 18731.8} C_VEL
LIN {X 0,Y 381.928,Z 85.584,A -85,B 0,C 180,E1 18728.506,E2 18728.506} C_VEL
LIN {X 0,Y 378.621,Z 77.654,A -85,B 0,C 180,E1 18726.064,E2 18726.064} C_VEL
LIN {X 0,Y 377.654,Z 74.858,A -85,B 0,C 180,E1 18725.089,E2 18725.089} C_VEL
LIN {X 0,Y 377.644,Z 74.755,A -85,B 0,C 180,E1 18721.062,E2 18721.062} C_VEL
LIN {X 0,Y 377.642,Z 74.757,A -85,B 0,C 180,E1 18717.117,E2 18717.117} C_VEL
LIN {X 0,Y 377.641,Z 74.758,A -85,B 0,C 180,E1 18713.153,E2 18713.153} C_VEL
LIN {X 0,Y 377.643,Z 74.757,A -85,B 0,C 180,E1 18709.165,E2 18709.165} C_VEL
LIN {X 0,Y 377.638,Z 74.755,A -85,B 0,C 180,E1 18705.276,E2 18705.276} C_VEL
LIN {X 0,Y 377.638,Z 74.752,A -85,B 0,C 180,E1 18701.315,E2 18701.315} C_VEL
LIN {X 0,Y 377.632,Z 74.755,A -85,B 0,C 180,E1 18697.424,E2 18697.424} C_VEL
LIN {X 0,Y 377.637,Z 74.755,A -85,B 0,C 180,E1 18693.42,E2 18693.42} C_VEL
LIN {X 0,Y 377.636,Z 74.755,A -85,B 0,C 180,E1 18689.446,E2 18689.446} C_VEL
LIN {X 0,Y 377.642,Z 74.755,A -85,B 0,C 180,E1 18685.429,E2 18685.429} C_VEL
LIN {X 0,Y 377.654,Z 74.758,A -85,B 0,C 180,E1 18681.331,E2 18681.331} C_VEL
LIN {X 0,Y 377.682,Z 75.018,A -85,B 0,C 180,E1 18678.912,E2 18678.912} C_VEL
LIN {X 0,Y 379.007,Z 78.367,A -85,B 0,C 180,E1 18677.927,E2 18677.927} C_VEL
LIN {X 0,Y 383.088,Z 87.34,A -85,B 0,C 180,E1 18675.51,E2 18675.51} C_VEL
LIN {X 0,Y 388.276,Z 100.025,A -85,B 0,C 180,E1 18672.567,E2 18672.567} C_VEL
LIN {X 0,Y 393.619,Z 114.916,A -85,B 0,C 180,E1 18669.612,E2 18669.612} C_VEL
LIN {X 0,Y 397.505,Z 127.592,A -85,B 0,C 180,E1 18667.406,E2 18667.406} C_VEL
LIN {X 0,Y 392.339,Z 162.109,A -85,B 0,C 180,E1 18663.542,E2 18663.542} C_VEL
LIN {X 0,Y 394.946,Z 186.381,A -85,B 0,C 180,E1 18662.775,E2 18662.775} C_VEL
LIN {X 0,Y 391.219,Z 353.49,A -85,B 0,C 180,E1 18659.662,E2 18659.662} C_VEL
LIN {X 0,Y 390.082,Z 371.882,A -85,B 0,C 180,E1 18659.069,E2 18659.069} C_VEL
LIN {X 0,Y 388.499,Z 389.656,A -85,B 0,C 180,E1 18658.227,E2 18658.227} C_VEL
LIN {X 0,Y 386.737,Z 406.483,A -85,B 0,C 180,E1 18657.151,E2 18657.151} C_VEL
LIN {X 0,Y 384.777,Z 422.977,A -85,B 0,C 180,E1 18655.802,E2 18655.802} C_VEL
LIN {X 0,Y 382.813,Z 438.574,A -85,B 0,C 180,E1 18654.21,E2 18654.21} C_VEL
LIN {X 0,Y 380.938,Z 453.253,A -85,B 0,C 180,E1 18652.371,E2 18652.371} C_VEL
LIN {X 0,Y 379.327,Z 466.468,A -85,B 0,C 180,E1 18650.362,E2 18650.362} C_VEL
LIN {X 0,Y 377.968,Z 479.087,A -85,B 0,C 180,E1 18648.03,E2 18648.03} C_VEL
LIN {X 0,Y 377.03,Z 490.131,A -85,B 0,C 180,E1 18645.537,E2 18645.537} C_VEL
LIN {X 0,Y 376.562,Z 499.333,A -85,B 0,C 180,E1 18642.975,E2 18642.975} C_VEL
LIN {X 0,Y 376.464,Z 507.067,A -85,B 0,C 180,E1 18640.251,E2 18640.251} C_VEL
LIN {X 0,Y 376.675,Z 512.993,A -85,B 0,C 180,E1 18637.475,E2 18637.475} C_VEL
LIN {X 0,Y 376.967,Z 516.837,A -85,B 0,C 180,E1 18634.87,E2 18634.87} C_VEL
LIN {X 0,Y 377.223,Z 519.104,A -85,B 0,C 180,E1 18632.195,E2 18632.195} C_VEL
LIN {X 0,Y 377.302,Z 519.681,A -85,B 0,C 180,E1 18629.697,E2 18629.697} C_VEL
LIN {X 0,Y 377.168,Z 518.697,A -85,B 0,C 180,E1 18627.114,E2 18627.114} C_VEL
LIN {X 0,Y 376.903,Z 516.094,A -85,B 0,C 180,E1 18624.521,E2 18624.521} C_VEL
LIN {X 0,Y 376.62,Z 511.814,A -85,B 0,C 180,E1 18621.913,E2 18621.913} C_VEL
LIN {X 0,Y 376.47,Z 505.767,A -85,B 0,C 180,E1 18619.287,E2 18619.287} C_VEL
LIN {X 0,Y 376.627,Z 497.8,A -85,B 0,C 180,E1 18616.648,E2 18616.648} C_VEL
LIN {X 0,Y 377.134,Z 488.326,A -85,B 0,C 180,E1 18614.154,E2 18614.154} C_VEL
LIN {X 0,Y 378.099,Z 476.748,A -85,B 0,C 180,E1 18611.686,E2 18611.686} C_VEL
LIN {X 0,Y 379.392,Z 464.116,A -85,B 0,C 180,E1 18609.483,E2 18609.483} C_VEL
LIN {X 0,Y 380.987,Z 450.096,A -85,B 0,C 180,E1 18607.472,E2 18607.472} C_VEL
LIN {X 0,Y 382.742,Z 435.115,A -85,B 0,C 180,E1 18605.714,E2 18605.714} C_VEL
LIN {X 0,Y 384.557,Z 418.945,A -85,B 0,C 180,E1 18604.184,E2 18604.184} C_VEL
LIN {X 0,Y 386.329,Z 401.831,A -85,B 0,C 180,E1 18602.904,E2 18602.904} C_VEL
LIN {X 0,Y 387.902,Z 384.307,A -85,B 0,C 180,E1 18601.903,E2 18601.903} C_VEL
LIN {X 0,Y 389.228,Z 365.467,A -85,B 0,C 180,E1 18601.136,E2 18601.136} C_VEL
LIN {X 0,Y 389.975,Z 346.9,A -85,B 0,C 180,E1 18600.655,E2 18600.655} C_VEL
LIN {X 0,Y 393.216,Z 173.183,A -85,B 0,C 180,E1 18597.498,E2 18597.498} C_VEL
LIN {X 0,Y 392.534,Z 157.215,A -85,B 0,C 180,E1 18597.101,E2 18597.101} C_VEL
LIN {X 0,Y 395.703,Z 119.168,A -85,B 0,C 180,E1 18594.701,E2 18594.701} C_VEL
LIN {X 0,Y 386.232,Z 95.124,A -85,B 0,C 180,E1 18592.145,E2 18592.145} C_VEL
LIN {X 0,Y 377.782,Z 75.334,A -85,B 0,C 180,E1 18589.778,E2 18589.778} C_VEL
LIN {X 0,Y 377.681,Z 74.752,A -85,B 0,C 180,E1 18589.446,E2 18589.446} C_VEL
LIN {X 0,Y 377.677,Z 74.751,A -85,B 0,C 180,E1 18585.41,E2 18585.41} C_VEL
LIN {X 0,Y 377.676,Z 74.747,A -85,B 0,C 180,E1 18581.239,E2 18581.239} C_VEL
LIN {X 0,Y 377.677,Z 74.753,A -85,B 0,C 180,E1 18577.172,E2 18577.172} C_VEL
LIN {X 0,Y 377.682,Z 74.751,A -85,B 0,C 180,E1 18573.049,E2 18573.049} C_VEL
LIN {X 0,Y 377.69,Z 74.749,A -85,B 0,C 180,E1 18568.977,E2 18568.977} C_VEL
LIN {X 0,Y 377.687,Z 74.751,A -85,B 0,C 180,E1 18564.893,E2 18564.893} C_VEL
LIN {X 0,Y 377.691,Z 74.752,A -85,B 0,C 180,E1 18560.777,E2 18560.777} C_VEL
LIN {X 0,Y 377.686,Z 74.754,A -85,B 0,C 180,E1 18556.605,E2 18556.605} C_VEL
LIN {X 0,Y 377.677,Z 74.752,A -85,B 0,C 180,E1 18552.538,E2 18552.538} C_VEL
LIN {X 0,Y 377.675,Z 74.745,A -85,B 0,C 180,E1 18548.526,E2 18548.526} C_VEL
LIN {X 0,Y 377.669,Z 74.741,A -85,B 0,C 180,E1 18544.555,E2 18544.555} C_VEL
LIN {X 0,Y 377.66,Z 74.742,A -85,B 0,C 180,E1 18540.455,E2 18540.455} C_VEL
LIN {X 0,Y 377.658,Z 74.75,A -85,B 0,C 180,E1 18536.357,E2 18536.357} C_VEL
LIN {X 0,Y 377.655,Z 74.753,A -85,B 0,C 180,E1 18532.24,E2 18532.24} C_VEL
LIN {X 0,Y 377.655,Z 74.753,A -85,B 0,C 180,E1 18528.237,E2 18528.237} C_VEL
LIN {X 0,Y 377.659,Z 74.752,A -85,B 0,C 180,E1 18524.175,E2 18524.175} C_VEL
LIN {X 0,Y 377.661,Z 74.753,A -85,B 0,C 180,E1 18520.191,E2 18520.191} C_VEL
LIN {X 0,Y 377.656,Z 74.717,A -85,B 0,C 180,E1 18516.27,E2 18516.27} C_VEL
LIN {X 0,Y 377.663,Z 74.754,A -85,B 0,C 180,E1 18512.227,E2 18512.227} C_VEL
LIN {X 0,Y 377.656,Z 74.742,A -85,B 0,C 180,E1 18508.384,E2 18508.384} C_VEL
LIN {X 0,Y 377.658,Z 74.734,A -85,B 0,C 180,E1 18504.366,E2 18504.366} C_VEL
LIN {X 0,Y 377.662,Z 74.742,A -85,B 0,C 180,E1 18500.353,E2 18500.353} C_VEL
LIN {X 0,Y 377.67,Z 74.741,A -85,B 0,C 180,E1 18496.291,E2 18496.291} C_VEL
LIN {X 0,Y 377.673,Z 74.962,A -85,B 0,C 180,E1 18492.871,E2 18492.871} C_VEL
LIN {X 0,Y 383.985,Z 93.031,A -85,B 0,C 180,E1 18490.026,E2 18490.026} C_VEL
LIN {X 0,Y 388.551,Z 109.089,A -85,B 0,C 180,E1 18487.693,E2 18487.693} C_VEL
LIN {X 0,Y 388.731,Z 113.823,A -85,B 0,C 180,E1 18487.121,E2 18487.121} C_VEL
LIN {X 0,Y 387.819,Z 148.123,A -85,B 0,C 180,E1 18483.13,E2 18483.13} C_VEL
LIN {X 0,Y 386.977,Z 183.944,A -85,B 0,C 180,E1 18479.06,E2 18479.06} C_VEL
LIN {X 0,Y 386.781,Z 199.962,A -85,B 0,C 180,E1 18477.339,E2 18477.339} C_VEL
LIN {X 0,Y 387.363,Z 204.94,A -85,B 0,C 180,E1 18477.197,E2 18477.197} C_VEL
LIN {X 0,Y 385.747,Z 307.37,A -85,B 0,C 180,E1 18475.264,E2 18475.264} C_VEL
LIN {X 0,Y 385.673,Z 322.164,A -85,B 0,C 180,E1 18474.801,E2 18474.801} C_VEL
LIN {X 0,Y 385.267,Z 336.211,A -85,B 0,C 180,E1 18474.097,E2 18474.097} C_VEL
LIN {X 0,Y 384.527,Z 349.948,A -85,B 0,C 180,E1 18473.117,E2 18473.117} C_VEL
LIN {X 0,Y 383.552,Z 362.789,A -85,B 0,C 180,E1 18471.885,E2 18471.885} C_VEL
LIN {X 0,Y 382.542,Z 373.973,A -85,B 0,C 180,E1 18470.5,E2 18470.5} C_VEL
LIN {X 0,Y 381.39,Z 384.649,A -85,B 0,C 180,E1 18468.81,E2 18468.81} C_VEL
LIN {X 0,Y 380.226,Z 394.305,A -85,B 0,C 180,E1 18466.812,E2 18466.812} C_VEL
LIN {X 0,Y 379.235,Z 402.069,A -85,B 0,C 180,E1 18464.66,E2 18464.66} C_VEL
LIN {X 0,Y 378.502,Z 407.625,A -85,B 0,C 180,E1 18462.509,E2 18462.509} C_VEL
LIN {X 0,Y 377.997,Z 411.337,A -85,B 0,C 180,E1 18460.361,E2 18460.361} C_VEL
LIN {X 0,Y 377.675,Z 413.49,A -85,B 0,C 180,E1 18458.053,E2 18458.053} C_VEL
LIN {X 0,Y 377.539,Z 413.773,A -85,B 0,C 180,E1 18455.622,E2 18455.622} C_VEL
LIN {X 0,Y 377.601,Z 412.032,A -85,B 0,C 180,E1 18453.186,E2 18453.186} C_VEL
LIN {X 0,Y 377.851,Z 408.5,A -85,B 0,C 180,E1 18450.909,E2 18450.909} C_VEL
LIN {X 0,Y 378.265,Z 403.408,A -85,B 0,C 180,E1 18448.787,E2 18448.787} C_VEL
LIN {X 0,Y 378.286,Z 403.154,A -85,B 0,C 180,E1 18448.7,E2 18448.7} C_VEL
LIN {X 0,Y 377.587,Z 400.012,A -85,B 0,C 180,E1 18447.63,E2 18447.63} C_VEL
LIN {X 0,Y 374.131,Z 394.156,A -85,B 0,C 180,E1 18445.866,E2 18445.866} C_VEL
LIN {X 0,Y 372.151,Z 388.899,A -85,B 0,C 180,E1 18444.588,E2 18444.588} C_VEL
LIN {X 0,Y 372.064,Z 386.159,A -85,B 0,C 180,E1 18444.043,E2 18444.043} C_VEL
LIN {X 0,Y 372.939,Z 376.045,A -85,B 0,C 180,E1 18442.373,E2 18442.373} C_VEL
LIN {X 0,Y 373.785,Z 364.892,A -85,B 0,C 180,E1 18440.918,E2 18440.918} C_VEL
LIN {X 0,Y 374.587,Z 351.947,A -85,B 0,C 180,E1 18439.619,E2 18439.619} C_VEL
LIN {X 0,Y 375.215,Z 338.73,A -85,B 0,C 180,E1 18438.626,E2 18438.626} C_VEL
LIN {X 0,Y 375.576,Z 324.5,A -85,B 0,C 180,E1 18437.858,E2 18437.858} C_VEL
LIN {X 0,Y 375.639,Z 309.079,A -85,B 0,C 180,E1 18437.341,E2 18437.341} C_VEL
LIN {X 0,Y 376.741,Z 222.093,A -85,B 0,C 180,E1 18435.678,E2 18435.678} C_VEL
LIN {X 0,Y 377.251,Z 196.728,A -85,B 0,C 180,E1 18435.18,E2 18435.18} C_VEL
LIN {X 0,Y 377.911,Z 187.379,A -85,B 0,C 180,E1 18434.579,E2 18434.579} C_VEL
LIN {X 0,Y 378.294,Z 174.193,A -85,B 0,C 180,E1 18433.65,E2 18433.65} C_VEL
LIN {X 0,Y 378.951,Z 172.937,A -85,B 0,C 180,E1 18433.364,E2 18433.364} C_VEL
LIN {X 0,Y 380.032,Z 173.432,A -85,B 0,C 180,E1 18433.177,E2 18433.177} C_VEL
LIN {X 0,Y 380.494,Z 174.4,A -85,B 0,C 180,E1 18433.114,E2 18433.114} C_VEL
LIN {X 0,Y 382.164,Z 196.314,A -85,B 0,C 180,E1 18432.486,E2 18432.486} C_VEL
LIN {X 0,Y 379.221,Z 300.523,A -85,B 0,C 180,E1 18430.201,E2 18430.201} C_VEL
LIN {X 0,Y 378.571,Z 317.401,A -85,B 0,C 180,E1 18429.536,E2 18429.536} C_VEL
LIN {X 0,Y 377.628,Z 333.057,A -85,B 0,C 180,E1 18428.613,E2 18428.613} C_VEL
LIN {X 0,Y 376.559,Z 346.902,A -85,B 0,C 180,E1 18427.519,E2 18427.519} C_VEL
LIN {X 0,Y 375.247,Z 361.184,A -85,B 0,C 180,E1 18426.056,E2 18426.056} C_VEL
LIN {X 0,Y 373.997,Z 373.409,A -85,B 0,C 180,E1 18424.442,E2 18424.442} C_VEL
LIN {X 0,Y 372.84,Z 383.954,A -85,B 0,C 180,E1 18422.704,E2 18422.704} C_VEL
LIN {X 0,Y 371.73,Z 393.811,A -85,B 0,C 180,E1 18420.632,E2 18420.632} C_VEL
LIN {X 0,Y 370.92,Z 401.119,A -85,B 0,C 180,E1 18418.65,E2 18418.65} C_VEL
LIN {X 0,Y 370.255,Z 407.671,A -85,B 0,C 180,E1 18416.279,E2 18416.279} C_VEL
LIN {X 0,Y 369.849,Z 412.121,A -85,B 0,C 180,E1 18413.889,E2 18413.889} C_VEL
LIN {X 0,Y 369.685,Z 414.697,A -85,B 0,C 180,E1 18411.532,E2 18411.532} C_VEL
LIN {X 0,Y 369.736,Z 415.481,A -85,B 0,C 180,E1 18408.981,E2 18408.981} C_VEL
LIN {X 0,Y 369.997,Z 414.415,A -85,B 0,C 180,E1 18406.63,E2 18406.63} C_VEL
LIN {X 0,Y 370.539,Z 411.348,A -85,B 0,C 180,E1 18404.122,E2 18404.122} C_VEL
LIN {X 0,Y 371.33,Z 406.444,A -85,B 0,C 180,E1 18401.766,E2 18401.766} C_VEL
LIN {X 0,Y 372.371,Z 400.064,A -85,B 0,C 180,E1 18399.589,E2 18399.589} C_VEL
LIN {X 0,Y 373.744,Z 391.367,A -85,B 0,C 180,E1 18397.394,E2 18397.394} C_VEL
LIN {X 0,Y 375.198,Z 381.766,A -85,B 0,C 180,E1 18395.518,E2 18395.518} C_VEL
LIN {X 0,Y 376.777,Z 370.493,A -85,B 0,C 180,E1 18393.777,E2 18393.777} C_VEL
LIN {X 0,Y 378.355,Z 357.994,A -85,B 0,C 180,E1 18392.258,E2 18392.258} C_VEL
LIN {X 0,Y 379.831,Z 344.482,A -85,B 0,C 180,E1 18390.964,E2 18390.964} C_VEL
LIN {X 0,Y 381.105,Z 329.883,A -85,B 0,C 180,E1 18389.9,E2 18389.9} C_VEL
LIN {X 0,Y 382.133,Z 314.392,A -85,B 0,C 180,E1 18389.067,E2 18389.067} C_VEL
LIN {X 0,Y 382.848,Z 297.217,A -85,B 0,C 180,E1 18388.466,E2 18388.466} C_VEL
LIN {X 0,Y 386.282,Z 206.169,A -85,B 0,C 180,E1 18386.292,E2 18386.292} C_VEL
LIN {X 0,Y 381.11,Z 177.087,A -85,B 0,C 180,E1 18385.007,E2 18385.007} C_VEL
LIN {X 0,Y 380.253,Z 172.459,A -85,B 0,C 180,E1 18384.756,E2 18384.756} C_VEL
LIN {X 0,Y 383.845,Z 145.359,A -85,B 0,C 180,E1 18380.43,E2 18380.43} C_VEL
LIN {X 0,Y 386.478,Z 127.215,A -85,B 0,C 180,E1 18377.464,E2 18377.464} C_VEL
LIN {X 0,Y 383.17,Z 113.903,A -85,B 0,C 180,E1 18374.508,E2 18374.508} C_VEL
LIN {X 0,Y 379.562,Z 101.858,A -85,B 0,C 180,E1 18371.549,E2 18371.549} C_VEL
LIN {X 0,Y 375.407,Z 90.037,A -85,B 0,C 180,E1 18368.27,E2 18368.27} C_VEL
LIN {X 0,Y 372.28,Z 82.393,A -85,B 0,C 180,E1 18365.858,E2 18365.858} C_VEL
LIN {X 0,Y 369.724,Z 75.879,A -85,B 0,C 180,E1 18363.566,E2 18363.566} C_VEL
LIN {X 0,Y 369.7,Z 75.744,A -85,B 0,C 180,E1 18359.535,E2 18359.535} C_VEL
LIN {X 0,Y 369.698,Z 75.746,A -85,B 0,C 180,E1 18355.346,E2 18355.346} C_VEL
